LIN {X -0.084,Y -142.879,Z 263.170,A 0.000,B 0.000,C 90.000,E1 210.669} C_DIS
LIN {X -0.027,Y -141.496,Z 263.150,A 0.000,B 0.000,C 90.000,E1 206.950} C_DIS
LIN {X 0.023,Y -139.387,Z 263.114,A 0.000,B 0.000,C 90.000,E1 200.429} C_DIS
LIN {X 0.010,Y -138.843,Z 263.098,A 0.000,B 0.000,C 90.000,E1 197.638} C_DIS
LIN {X -0.066,Y -138.354,Z 263.056,A 0.000,B 0.000,C 90.000,E1 190.197} C_DIS
LIN {X 0.067,Y -139.519,Z 263.005,A 0.000,B 0.000,C 90.000,E1 180.802} C_DIS
LIN {X 0.007,Y -141.176,Z 262.974,A 0.000,B 0.000,C 90.000,E1 175.241} C_DIS
LIN {X -0.021,Y -142.555,Z 262.958,A 0.000,B 0.000,C 90.000,E1 172.470} C_DIS
LIN {X 0.046,Y -144.834,Z 262.932,A 0.000,B 0.000,C 90.000,E1 167.825} C_DIS
LIN {X 0.031,Y -147.457,Z 262.912,A 0.000,B 0.000,C 90.000,E1 164.157} C_DIS
LIN {X -0.082,Y -150.039,Z 262.892,A 0.000,B 0.000,C 90.000,E1 160.550} C_DIS
LIN {X -0.076,Y -153.380,Z 262.872,A 0.000,B 0.000,C 90.000,E1 156.922} C_DIS
LIN {X -0.029,Y -155.912,Z 262.857,A 0.000,B 0.000,C 90.000,E1 154.204} C_DIS
LIN {X 0.087,Y -159.775,Z 262.837,A 0.000,B 0.000,C 90.000,E1 150.589} C_DIS
LIN {X -0.066,Y -162.015,Z 262.827,A 0.000,B 0.000,C 90.000,E1 148.869} C_DIS
LIN {X 0.048,Y -166.209,Z 262.807,A 0.000,B 0.000,C 90.000,E1 145.308} C_DIS
LIN {X 0.049,Y -171.225,Z 262.788,A 0.000,B 0.000,C 90.000,E1 141.823} C_DIS
LIN {X -0.026,Y -176.111,Z 262.769,A 0.000,B 0.000,C 90.000,E1 138.405} C_DIS
LIN {X 0.090,Y -180.375,Z 262.755,A 0.000,B 0.000,C 90.000,E1 135.810} C_DIS
LIN {X 0.067,Y -185.783,Z 262.736,A 0.000,B 0.000,C 90.000,E1 132.447} C_DIS
LIN {X 0.000,Y -190.399,Z 262.722,A 0.000,B 0.000,C 90.000,E1 129.967} C_DIS
LIN {X 0.016,Y -197.723,Z 262.699,A 0.000,B 0.000,C 90.000,E1 125.851} C_DIS
LIN {X -0.060,Y -200.971,Z 262.690,A 0.000,B 0.000,C 90.000,E1 124.246} C_DIS
LIN {X 0.078,Y -203.895,Z 262.681,A 0.000,B 0.000,C 90.000,E1 122.546} C_DIS
LIN {X 0.064,Y -306.288,Z 262.681,A 0.000,B 0.000,C 90.000,E1 122.546} C_DIS
LIN {X 0.009,Y -307.336,Z 262.681,A 0.000,B 0.000,C 90.000,E1 122.546} C_DIS
LIN {X 0.131,Y -312.237,Z 262.680,A 0.000,B 0.000,C 90.000,E1 122.339} C_DIS
LIN {X -0.178,Y -314.694,Z 262.679,A 0.000,B 0.000,C 90.000,E1 122.212} C_DIS
LIN {X 0.068,Y -318.006,Z 262.677,A 0.000,B 0.000,C 90.000,E1 121.799} C_DIS
LIN {X -0.031,Y -319.961,Z 262.675,A 0.000,B 0.000,C 90.000,E1 121.514} C_DIS
LIN {X -0.026,Y -321.496,Z 262.673,A 0.000,B 0.000,C 90.000,E1 121.209} C_DIS
LIN {X 0.054,Y -335.561,Z 262.654,A 0.000,B 0.000,C 90.000,E1 117.719} C_DIS
LIN {X -0.033,Y -348.593,Z 262.639,A 0.000,B 0.000,C 90.000,E1 114.951} C_DIS
LIN {X 0.068,Y -361.495,Z 262.625,A 0.000,B 0.000,C 90.000,E1 112.514} C_DIS
LIN {X -0.119,Y -375.736,Z 262.612,A 0.000,B 0.000,C 90.000,E1 110.174} C_DIS
LIN {X 0.152,Y -391.421,Z 262.599,A 0.000,B 0.000,C 90.000,E1 107.819} C_DIS
LIN {X -0.164,Y -408.665,Z 262.587,A 0.000,B 0.000,C 90.000,E1 105.607} C_DIS
LIN {X -0.185,Y -427.600,Z 262.574,A 0.000,B 0.000,C 90.000,E1 103.411} C_DIS
LIN {X 0.123,Y -447.711,Z 262.563,A 0.000,B 0.000,C 90.000,E1 101.299} C_DIS
LIN {X -0.145,Y -468.376,Z 262.552,A 0.000,B 0.000,C 90.000,E1 99.434} C_DIS
LIN {X 0.024,Y -492.186,Z 262.542,A 0.000,B 0.000,C 90.000,E1 97.466} C_DIS
LIN {X -0.023,Y -502.840,Z 262.537,A 0.000,B 0.000,C 90.000,E1 96.663} C_DIS
LIN {X -0.205,Y -504.840,Z 262.536,A 0.000,B 0.000,C 90.000,E1 96.486} C_DIS
LIN {X 0.199,Y -506.671,Z 262.535,A 0.000,B 0.000,C 90.000,E1 96.201} C_DIS
LIN {X 0.157,Y -508.048,Z 262.533,A 0.000,B 0.000,C 90.000,E1 95.967} C_DIS
LIN {X -0.073,Y -509.799,Z 262.531,A 0.000,B 0.000,C 90.000,E1 95.511} C_DIS
LIN {X -0.244,Y -510.440,Z 262.528,A 0.000,B 0.000,C 90.000,E1 95.049} C_DIS
LIN {X 0.101,Y -510.071,Z 262.525,A 0.000,B 0.000,C 90.000,E1 94.531} C_DIS
LIN {X -0.099,Y -508.627,Z 262.523,A 0.000,B 0.000,C 90.000,E1 94.073} C_DIS
LIN {X -0.163,Y -507.423,Z 262.521,A 0.000,B 0.000,C 90.000,E1 93.841} C_DIS
LIN {X 0.138,Y -503.972,Z 262.519,A 0.000,B 0.000,C 90.000,E1 93.326} C_DIS
LIN {X -0.166,Y -498.128,Z 262.515,A 0.000,B 0.000,C 90.000,E1 92.636} C_DIS
LIN {X 0.187,Y -487.577,Z 262.508,A 0.000,B 0.000,C 90.000,E1 91.375} C_DIS
LIN {X -0.069,Y -466.396,Z 262.494,A 0.000,B 0.000,C 90.000,E1 88.912} C_DIS
LIN {X 0.086,Y -451.279,Z 262.483,A 0.000,B 0.000,C 90.000,E1 86.846} C_DIS
LIN {X 0.022,Y -432.472,Z 262.467,A 0.000,B 0.000,C 90.000,E1 83.970} C_DIS
LIN {X 0.219,Y -416.903,Z 262.452,A 0.000,B 0.000,C 90.000,E1 81.254} C_DIS
LIN {X -0.015,Y -404.099,Z 262.438,A 0.000,B 0.000,C 90.000,E1 78.814} C_DIS
LIN {X -0.040,Y -391.301,Z 262.424,A 0.000,B 0.000,C 90.000,E1 76.297} C_DIS
LIN {X -0.128,Y -378.784,Z 262.410,A 0.000,B 0.000,C 90.000,E1 73.740} C_DIS
LIN {X -0.060,Y -367.611,Z 262.397,A 0.000,B 0.000,C 90.000,E1 71.402} C_DIS
LIN {X -0.032,Y -356.629,Z 262.383,A 0.000,B 0.000,C 90.000,E1 69.028} C_DIS
LIN {X 0.187,Y -342.383,Z 262.365,A 0.000,B 0.000,C 90.000,E1 65.665} C_DIS
LIN {X -0.064,Y -330.397,Z 262.348,A 0.000,B 0.000,C 90.000,E1 62.615} C_DIS
LIN {X -0.055,Y -319.220,Z 262.330,A 0.000,B 0.000,C 90.000,E1 59.459} C_DIS
LIN {X -0.178,Y -310.444,Z 262.316,A 0.000,B 0.000,C 90.000,E1 56.914} C_DIS
LIN {X -0.009,Y -299.955,Z 262.298,A 0.000,B 0.000,C 90.000,E1 53.623} C_DIS
LIN {X 0.093,Y -293.735,Z 262.287,A 0.000,B 0.000,C 90.000,E1 51.618} C_DIS
LIN {X 0.103,Y -285.428,Z 262.272,A 0.000,B 0.000,C 90.000,E1 48.933} C_DIS
LIN {X -0.121,Y -275.297,Z 262.253,A 0.000,B 0.000,C 90.000,E1 45.567} C_DIS
LIN {X -0.020,Y -267.641,Z 262.238,A 0.000,B 0.000,C 90.000,E1 42.771} C_DIS
LIN {X 0.090,Y -260.135,Z 262.222,A 0.000,B 0.000,C 90.000,E1 39.930} C_DIS
LIN {X 0.007,Y -254.382,Z 262.210,A 0.000,B 0.000,C 90.000,E1 37.810} C_DIS
LIN {X 0.016,Y -248.606,Z 262.198,A 0.000,B 0.000,C 90.000,E1 35.644} C_DIS
LIN {X -0.117,Y -240.937,Z 262.182,A 0.000,B 0.000,C 90.000,E1 32.752} C_DIS
LIN {X 0.033,Y -231.734,Z 262.161,A 0.000,B 0.000,C 90.000,E1 28.999} C_DIS
LIN {X 0.028,Y -225.126,Z 262.144,A 0.000,B 0.000,C 90.000,E1 25.976} C_DIS
LIN {X 0.076,Y -219.297,Z 262.127,A 0.000,B 0.000,C 90.000,E1 22.898} C_DIS
LIN {X 0.002,Y -212.842,Z 262.106,A 0.000,B 0.000,C 90.000,E1 19.033} C_DIS
LIN {X 0.068,Y -207.446,Z 262.084,A 0.000,B 0.000,C 90.000,E1 15.079} C_DIS
LIN {X -0.045,Y -202.998,Z 262.062,A 0.000,B 0.000,C 90.000,E1 11.130} C_DIS
LIN {X -0.087,Y -199.578,Z 262.039,A 0.000,B 0.000,C 90.000,E1 7.125} C_DIS
LIN {X -0.009,Y -196.386,Z 262.008,A 0.000,B 0.000,C 90.000,E1 1.432} C_DIS
LIN {X 0.078,Y -197.440,Z 261.920,A 0.000,B 0.000,C 90.000,E1 345.644} C_DIS
LIN {X 0.059,Y -200.766,Z 261.893,A 0.000,B 0.000,C 90.000,E1 340.786} C_DIS
LIN {X -0.056,Y -204.789,Z 261.871,A 0.000,B 0.000,C 90.000,E1 336.794} C_DIS
LIN {X -0.009,Y -209.928,Z 261.849,A 0.000,B 0.000,C 90.000,E1 332.794} C_DIS
LIN {X -0.070,Y -216.233,Z 261.827,A 0.000,B 0.000,C 90.000,E1 328.869} C_DIS
LIN {X 0.059,Y -222.165,Z 261.810,A 0.000,B 0.000,C 90.000,E1 325.722} C_DIS
LIN {X 0.102,Y -228.969,Z 261.793,A 0.000,B 0.000,C 90.000,E1 322.637} C_DIS
LIN {X 0.006,Y -237.487,Z 261.774,A 0.000,B 0.000,C 90.000,E1 319.256} C_DIS
LIN {X 0.112,Y -246.994,Z 261.755,A 0.000,B 0.000,C 90.000,E1 315.891} C_DIS
LIN {X 0.155,Y -257.496,Z 261.737,A 0.000,B 0.000,C 90.000,E1 312.609} C_DIS
LIN {X -0.005,Y -269.138,Z 261.719,A 0.000,B 0.000,C 90.000,E1 309.439} C_DIS
LIN {X 0.042,Y -282.107,Z 261.702,A 0.000,B 0.000,C 90.000,E1 306.297} C_DIS
LIN {X 0.039,Y -295.069,Z 261.687,A 0.000,B 0.000,C 90.000,E1 303.579} C_DIS
LIN {X -0.016,Y -305.748,Z 261.676,A 0.000,B 0.000,C 90.000,E1 301.592} C_DIS
LIN {X -0.065,Y -321.117,Z 261.661,A 0.000,B 0.000,C 90.000,E1 298.999} C_DIS
LIN {X -0.072,Y -339.487,Z 261.645,A 0.000,B 0.000,C 90.000,E1 296.155} C_DIS
LIN {X 0.084,Y -351.911,Z 261.635,A 0.000,B 0.000,C 90.000,E1 294.283} C_DIS
LIN {X 0.167,Y -364.417,Z 261.625,A 0.000,B 0.000,C 90.000,E1 292.461} C_DIS
LIN {X 0.079,Y -381.335,Z 261.612,A 0.000,B 0.000,C 90.000,E1 290.120} C_DIS
LIN {X -0.025,Y -396.501,Z 261.601,A 0.000,B 0.000,C 90.000,E1 288.127} C_DIS
LIN {X -0.114,Y -407.339,Z 261.593,A 0.000,B 0.000,C 90.000,E1 286.732} C_DIS
LIN {X 0.095,Y -422.232,Z 261.582,A 0.000,B 0.000,C 90.000,E1 284.773} C_DIS
LIN {X -0.012,Y -430.385,Z 261.576,A 0.000,B 0.000,C 90.000,E1 283.703} C_DIS
LIN {X -0.129,Y -437.902,Z 261.570,A 0.000,B 0.000,C 90.000,E1 282.647} C_DIS
LIN {X -0.159,Y -444.744,Z 261.564,A 0.000,B 0.000,C 90.000,E1 281.591} C_DIS
LIN {X -0.144,Y -454.217,Z 261.556,A 0.000,B 0.000,C 90.000,E1 280.018} C_DIS
LIN {X 0.138,Y -461.619,Z 261.548,A 0.000,B 0.000,C 90.000,E1 278.690} C_DIS
LIN {X 0.150,Y -468.491,Z 261.541,A 0.000,B 0.000,C 90.000,E1 277.409} C_DIS
LIN {X -0.133,Y -473.614,Z 261.536,A 0.000,B 0.000,C 90.000,E1 276.429} C_DIS
LIN {X -0.217,Y -477.139,Z 261.531,A 0.000,B 0.000,C 90.000,E1 275.682} C_DIS
LIN {X -0.079,Y -479.157,Z 261.529,A 0.000,B 0.000,C 90.000,E1 275.163} C_DIS
LIN {X 0.065,Y -480.938,Z 261.526,A 0.000,B 0.000,C 90.000,E1 274.645} C_DIS
LIN {X 0.185,Y -482.344,Z 261.523,A 0.000,B 0.000,C 90.000,E1 274.131} C_DIS
LIN {X -0.132,Y -483.499,Z 261.520,A 0.000,B 0.000,C 90.000,E1 273.669} C_DIS
LIN {X 0.012,Y -484.296,Z 261.518,A 0.000,B 0.000,C 90.000,E1 273.154} C_DIS
LIN {X 0.188,Y -484.741,Z 261.515,A 0.000,B 0.000,C 90.000,E1 272.636} C_DIS
LIN {X 0.041,Y -485.008,Z 261.509,A 0.000,B 0.000,C 90.000,E1 271.661} C_DIS
LIN {X 0.203,Y -484.935,Z 261.507,A 0.000,B 0.000,C 90.000,E1 271.146} C_DIS
LIN {X -0.117,Y -484.681,Z 261.504,A 0.000,B 0.000,C 90.000,E1 270.688} C_DIS
LIN {X 0.049,Y -484.046,Z 261.501,A 0.000,B 0.000,C 90.000,E1 270.172} C_DIS
LIN {X 0.212,Y -483.060,Z 261.498,A 0.000,B 0.000,C 90.000,E1 269.656} C_DIS
LIN {X -0.112,Y -481.501,Z 261.495,A 0.000,B 0.000,C 90.000,E1 269.198} C_DIS
LIN {X 0.040,Y -479.301,Z 261.493,A 0.000,B 0.000,C 90.000,E1 268.682} C_DIS
LIN {X 0.175,Y -476.392,Z 261.490,A 0.000,B 0.000,C 90.000,E1 268.167} C_DIS
LIN {X -0.164,Y -472.714,Z 261.487,A 0.000,B 0.000,C 90.000,E1 267.707} C_DIS
LIN {X -0.063,Y -468.210,Z 261.484,A 0.000,B 0.000,C 90.000,E1 267.192} C_DIS
LIN {X 0.205,Y -465.592,Z 261.483,A 0.000,B 0.000,C 90.000,E1 266.906} C_DIS
LIN {X 0.034,Y -462.649,Z 261.482,A 0.000,B 0.000,C 90.000,E1 266.674} C_DIS
LIN {X 0.083,Y -456.463,Z 261.479,A 0.000,B 0.000,C 90.000,E1 266.216} C_DIS
LIN {X -0.104,Y -453.228,Z 261.478,A 0.000,B 0.000,C 90.000,E1 266.045} C_DIS
LIN {X 0.193,Y -449.532,Z 261.477,A 0.000,B 0.000,C 90.000,E1 265.812} C_DIS
LIN {X -0.132,Y -445.984,Z 261.476,A 0.000,B 0.000,C 90.000,E1 265.698} C_DIS
LIN {X -0.011,Y -441.741,Z 261.475,A 0.000,B 0.000,C 90.000,E1 265.527} C_DIS
LIN {X -0.002,Y -437.789,Z 261.475,A 0.000,B 0.000,C 90.000,E1 265.412} C_DIS
LIN {X 0.008,Y -432.446,Z 261.474,A 0.000,B 0.000,C 90.000,E1 265.298} C_DIS
LIN {X 0.144,Y -425.453,Z 261.473,A 0.000,B 0.000,C 90.000,E1 265.179} C_DIS
LIN {X -0.163,Y -418.203,Z 261.473,A 0.000,B 0.000,C 90.000,E1 265.179} C_DIS
LIN {X 0.084,Y -180.889,Z 261.473,A 0.000,B 0.000,C 90.000,E1 265.122} C_DIS
LIN {X -0.014,Y -179.001,Z 261.445,A 0.000,B 0.000,C 90.000,E1 260.038} C_DIS
LIN {X 0.079,Y -178.598,Z 261.440,A 0.000,B 0.000,C 90.000,E1 259.162} C_DIS
LIN {X -0.027,Y -175.650,Z 261.412,A 0.000,B 0.000,C 90.000,E1 254.102} C_DIS
LIN {X -0.021,Y -172.368,Z 261.388,A 0.000,B 0.000,C 90.000,E1 249.826} C_DIS
LIN {X -0.007,Y -171.160,Z 261.378,A 0.000,B 0.000,C 90.000,E1 248.103} C_DIS
LIN {X 0.037,Y -167.459,Z 261.354,A 0.000,B 0.000,C 90.000,E1 243.768} C_DIS
LIN {X -0.030,Y -166.856,Z 261.350,A 0.000,B 0.000,C 90.000,E1 242.922} C_DIS
LIN {X 0.035,Y -162.841,Z 261.325,A 0.000,B 0.000,C 90.000,E1 238.535} C_DIS
LIN {X 0.010,Y -161.524,Z 261.315,A 0.000,B 0.000,C 90.000,E1 236.786} C_DIS
LIN {X 0.050,Y -157.524,Z 261.291,A 0.000,B 0.000,C 90.000,E1 232.351} C_DIS
LIN {X -0.017,Y -155.548,Z 261.276,A 0.000,B 0.000,C 90.000,E1 229.703} C_DIS
LIN {X -0.082,Y -151.840,Z 261.251,A 0.000,B 0.000,C 90.000,E1 225.243} C_DIS
LIN {X -0.068,Y -150.058,Z 261.236,A 0.000,B 0.000,C 90.000,E1 222.528} C_DIS
LIN {X -0.033,Y -146.870,Z 261.211,A 0.000,B 0.000,C 90.000,E1 217.971} C_DIS
LIN {X -0.044,Y -145.455,Z 261.196,A 0.000,B 0.000,C 90.000,E1 215.231} C_DIS
LIN {X 0.070,Y -142.871,Z 261.170,A 0.000,B 0.000,C 90.000,E1 210.590} C_DIS
LIN {X -0.005,Y -141.489,Z 261.150,A 0.000,B 0.000,C 90.000,E1 206.924} C_DIS
LIN {X -0.020,Y -139.384,Z 261.113,A 0.000,B 0.000,C 90.000,E1 200.429} C_DIS
LIN {X -0.031,Y -138.839,Z 261.098,A 0.000,B 0.000,C 90.000,E1 197.638} C_DIS
LIN {X 0.029,Y -138.353,Z 261.056,A 0.000,B 0.000,C 90.000,E1 190.141} C_DIS
LIN {X 0.025,Y -139.521,Z 261.005,A 0.000,B 0.000,C 90.000,E1 180.802} C_DIS
LIN {X -0.035,Y -141.184,Z 260.973,A 0.000,B 0.000,C 90.000,E1 175.241} C_DIS
LIN {X -0.064,Y -142.562,Z 260.958,A 0.000,B 0.000,C 90.000,E1 172.470} C_DIS
LIN {X 0.002,Y -144.844,Z 260.932,A 0.000,B 0.000,C 90.000,E1 167.825} C_DIS
LIN {X -0.012,Y -147.469,Z 260.912,A 0.000,B 0.000,C 90.000,E1 164.157} C_DIS
LIN {X 0.016,Y -150.054,Z 260.892,A 0.000,B 0.000,C 90.000,E1 160.496} C_DIS
LIN {X 0.020,Y -153.397,Z 260.872,A 0.000,B 0.000,C 90.000,E1 156.869} C_DIS
LIN {X 0.067,Y -155.927,Z 260.857,A 0.000,B 0.000,C 90.000,E1 154.152} C_DIS
LIN {X 0.041,Y -159.795,Z 260.837,A 0.000,B 0.000,C 90.000,E1 150.589} C_DIS
LIN {X 0.026,Y -162.035,Z 260.827,A 0.000,B 0.000,C 90.000,E1 148.820} C_DIS
LIN {X 0.001,Y -166.231,Z 260.807,A 0.000,B 0.000,C 90.000,E1 145.308} C_DIS
LIN {X 0.002,Y -171.247,Z 260.788,A 0.000,B 0.000,C 90.000,E1 141.823} C_DIS
LIN {X -0.075,Y -176.136,Z 260.769,A 0.000,B 0.000,C 90.000,E1 138.405} C_DIS
LIN {X 0.041,Y -180.403,Z 260.755,A 0.000,B 0.000,C 90.000,E1 135.810} C_DIS
LIN {X 0.017,Y -185.810,Z 260.736,A 0.000,B 0.000,C 90.000,E1 132.447} C_DIS
LIN {X 0.071,Y -190.429,Z 260.722,A 0.000,B 0.000,C 90.000,E1 129.930} C_DIS
LIN {X -0.037,Y -197.753,Z 260.699,A 0.000,B 0.000,C 90.000,E1 125.851} C_DIS
LIN {X 0.054,Y -200.996,Z 260.690,A 0.000,B 0.000,C 90.000,E1 124.199} C_DIS
LIN {X 0.031,Y -204.009,Z 260.681,A 0.000,B 0.000,C 90.000,E1 122.498} C_DIS
LIN {X -0.005,Y -307.390,Z 260.681,A 0.000,B 0.000,C 90.000,E1 122.498} C_DIS
LIN {X 0.002,Y -308.854,Z 260.680,A 0.000,B 0.000,C 90.000,E1 122.467} C_DIS
LIN {X 0.047,Y -312.597,Z 260.679,A 0.000,B 0.000,C 90.000,E1 122.291} C_DIS
LIN {X -0.007,Y -314.817,Z 260.678,A 0.000,B 0.000,C 90.000,E1 122.133} C_DIS
LIN {X -0.014,Y -317.903,Z 260.677,A 0.000,B 0.000,C 90.000,E1 121.799} C_DIS
LIN {X 0.186,Y -319.892,Z 260.675,A 0.000,B 0.000,C 90.000,E1 121.465} C_DIS
LIN {X -0.052,Y -321.453,Z 260.673,A 0.000,B 0.000,C 90.000,E1 121.209} C_DIS
LIN {X -0.175,Y -331.546,Z 260.659,A 0.000,B 0.000,C 90.000,E1 118.693} C_DIS
LIN {X 0.085,Y -344.080,Z 260.644,A 0.000,B 0.000,C 90.000,E1 115.848} C_DIS
LIN {X -0.106,Y -356.507,Z 260.630,A 0.000,B 0.000,C 90.000,E1 113.439} C_DIS
LIN {X -0.080,Y -370.235,Z 260.617,A 0.000,B 0.000,C 90.000,E1 111.046} C_DIS
LIN {X -0.180,Y -385.367,Z 260.604,A 0.000,B 0.000,C 90.000,E1 108.725} C_DIS
LIN {X -0.156,Y -402.016,Z 260.591,A 0.000,B 0.000,C 90.000,E1 106.441} C_DIS
LIN {X 0.071,Y -420.304,Z 260.579,A 0.000,B 0.000,C 90.000,E1 104.189} C_DIS
LIN {X 0.030,Y -440.104,Z 260.567,A 0.000,B 0.000,C 90.000,E1 102.063} C_DIS
LIN {X 0.173,Y -460.571,Z 260.556,A 0.000,B 0.000,C 90.000,E1 100.084} C_DIS
LIN {X -0.112,Y -484.215,Z 260.545,A 0.000,B 0.000,C 90.000,E1 98.106} C_DIS
LIN {X -0.058,Y -502.890,Z 260.537,A 0.000,B 0.000,C 90.000,E1 96.663} C_DIS
LIN {X 0.262,Y -504.933,Z 260.536,A 0.000,B 0.000,C 90.000,E1 96.429} C_DIS
LIN {X 0.192,Y -506.782,Z 260.535,A 0.000,B 0.000,C 90.000,E1 96.201} C_DIS
LIN {X 0.176,Y -508.177,Z 260.533,A 0.000,B 0.000,C 90.000,E1 95.967} C_DIS
LIN {X -0.053,Y -509.984,Z 260.531,A 0.000,B 0.000,C 90.000,E1 95.511} C_DIS
LIN {X -0.224,Y -510.666,Z 260.528,A 0.000,B 0.000,C 90.000,E1 95.049} C_DIS
LIN {X 0.122,Y -510.338,Z 260.525,A 0.000,B 0.000,C 90.000,E1 94.531} C_DIS
LIN {X -0.077,Y -508.947,Z 260.523,A 0.000,B 0.000,C 90.000,E1 94.073} C_DIS
LIN {X -0.140,Y -507.775,Z 260.521,A 0.000,B 0.000,C 90.000,E1 93.841} C_DIS
LIN {X 0.163,Y -504.368,Z 260.519,A 0.000,B 0.000,C 90.000,E1 93.326} C_DIS
LIN {X -0.138,Y -498.540,Z 260.515,A 0.000,B 0.000,C 90.000,E1 92.636} C_DIS
LIN {X -0.127,Y -490.145,Z 260.509,A 0.000,B 0.000,C 90.000,E1 91.661} C_DIS
LIN {X -0.026,Y -466.770,Z 260.494,A 0.000,B 0.000,C 90.000,E1 88.912} C_DIS
LIN {X -0.107,Y -453.453,Z 260.484,A 0.000,B 0.000,C 90.000,E1 87.135} C_DIS
LIN {X 0.164,Y -436.097,Z 260.470,A 0.000,B 0.000,C 90.000,E1 84.489} C_DIS
LIN {X 0.134,Y -418.677,Z 260.453,A 0.000,B 0.000,C 90.000,E1 81.546} C_DIS
LIN {X 0.055,Y -404.388,Z 260.438,A 0.000,B 0.000,C 90.000,E1 78.814} C_DIS
LIN {X 0.036,Y -391.568,Z 260.424,A 0.000,B 0.000,C 90.000,E1 76.297} C_DIS
LIN {X -0.047,Y -379.079,Z 260.410,A 0.000,B 0.000,C 90.000,E1 73.740} C_DIS
LIN {X 0.026,Y -367.931,Z 260.397,A 0.000,B 0.000,C 90.000,E1 71.402} C_DIS
LIN {X 0.059,Y -356.974,Z 260.384,A 0.000,B 0.000,C 90.000,E1 69.028} C_DIS
LIN {X -0.026,Y -342.765,Z 260.365,A 0.000,B 0.000,C 90.000,E1 65.717} C_DIS
LIN {X 0.043,Y -330.801,Z 260.348,A 0.000,B 0.000,C 90.000,E1 62.615} C_DIS
LIN {X 0.067,Y -319.624,Z 260.330,A 0.000,B 0.000,C 90.000,E1 59.459} C_DIS
LIN {X -0.022,Y -310.881,Z 260.316,A 0.000,B 0.000,C 90.000,E1 56.914} C_DIS
LIN {X 0.154,Y -300.371,Z 260.298,A 0.000,B 0.000,C 90.000,E1 53.623} C_DIS
LIN {X 0.030,Y -294.159,Z 260.287,A 0.000,B 0.000,C 90.000,E1 51.662} C_DIS
LIN {X -0.127,Y -285.836,Z 260.272,A 0.000,B 0.000,C 90.000,E1 49.013} C_DIS
LIN {X 0.059,Y -275.703,Z 260.253,A 0.000,B 0.000,C 90.000,E1 45.567} C_DIS
LIN {X -0.033,Y -268.039,Z 260.238,A 0.000,B 0.000,C 90.000,E1 42.813} C_DIS
LIN {X -0.087,Y -260.528,Z 260.222,A 0.000,B 0.000,C 90.000,E1 40.011} C_DIS
LIN {X -0.002,Y -254.769,Z 260.210,A 0.000,B 0.000,C 90.000,E1 37.855} C_DIS
LIN {X -0.049,Y -247.083,Z 260.194,A 0.000,B 0.000,C 90.000,E1 34.978} C_DIS
LIN {X 0.121,Y -239.463,Z 260.178,A 0.000,B 0.000,C 90.000,E1 32.005} C_DIS
LIN {X -0.080,Y -232.152,Z 260.161,A 0.000,B 0.000,C 90.000,E1 29.077} C_DIS
LIN {X 0.033,Y -225.527,Z 260.145,A 0.000,B 0.000,C 90.000,E1 26.027} C_DIS
LIN {X 0.085,Y -219.685,Z 260.128,A 0.000,B 0.000,C 90.000,E1 22.950} C_DIS
LIN {X 0.018,Y -213.215,Z 260.106,A 0.000,B 0.000,C 90.000,E1 19.087} C_DIS
LIN {X -0.110,Y -207.817,Z 260.084,A 0.000,B 0.000,C 90.000,E1 15.190} C_DIS
LIN {X -0.015,Y -203.339,Z 260.062,A 0.000,B 0.000,C 90.000,E1 11.186} C_DIS
LIN {X -0.050,Y -199.886,Z 260.040,A 0.000,B 0.000,C 90.000,E1 7.182} C_DIS
LIN {X 0.003,Y -196.350,Z 260.004,A 0.000,B 0.000,C 90.000,E1 0.688} C_DIS
LIN {X 0.080,Y -197.248,Z 259.925,A 0.000,B 0.000,C 90.000,E1 346.464} C_DIS
LIN {X -0.061,Y -200.306,Z 259.898,A 0.000,B 0.000,C 90.000,E1 341.638} C_DIS
LIN {X -0.001,Y -204.069,Z 259.876,A 0.000,B 0.000,C 90.000,E1 337.592} C_DIS
LIN {X 0.035,Y -208.988,Z 259.853,A 0.000,B 0.000,C 90.000,E1 333.589} C_DIS
LIN {X -0.061,Y -215.090,Z 259.831,A 0.000,B 0.000,C 90.000,E1 329.665} C_DIS
LIN {X 0.104,Y -220.800,Z 259.814,A 0.000,B 0.000,C 90.000,E1 326.501} C_DIS
LIN {X 0.111,Y -227.432,Z 259.797,A 0.000,B 0.000,C 90.000,E1 323.417} C_DIS
LIN {X -0.133,Y -234.790,Z 259.780,A 0.000,B 0.000,C 90.000,E1 320.436} C_DIS
LIN {X -0.107,Y -243.924,Z 259.761,A 0.000,B 0.000,C 90.000,E1 317.067} C_DIS
LIN {X 0.015,Y -254.095,Z 259.743,A 0.000,B 0.000,C 90.000,E1 313.743} C_DIS
LIN {X -0.092,Y -265.335,Z 259.725,A 0.000,B 0.000,C 90.000,E1 310.539} C_DIS
LIN {X 0.001,Y -277.812,Z 259.708,A 0.000,B 0.000,C 90.000,E1 307.363} C_DIS
LIN {X 0.078,Y -288.604,Z 259.694,A 0.000,B 0.000,C 90.000,E1 304.945} C_DIS
LIN {X -0.086,Y -302.262,Z 259.679,A 0.000,B 0.000,C 90.000,E1 302.291} C_DIS
LIN {X 0.000,Y -319.334,Z 259.663,A 0.000,B 0.000,C 90.000,E1 299.333} C_DIS
LIN {X 0.079,Y -339.615,Z 259.645,A 0.000,B 0.000,C 90.000,E1 296.155} C_DIS
LIN {X -0.078,Y -352.006,Z 259.635,A 0.000,B 0.000,C 90.000,E1 294.335} C_DIS
LIN {X -0.004,Y -364.464,Z 259.625,A 0.000,B 0.000,C 90.000,E1 292.514} C_DIS
LIN {X -0.104,Y -381.346,Z 259.612,A 0.000,B 0.000,C 90.000,E1 290.174} C_DIS
LIN {X -0.054,Y -398.637,Z 259.599,A 0.000,B 0.000,C 90.000,E1 287.873} C_DIS
LIN {X 0.163,Y -409.395,Z 259.591,A 0.000,B 0.000,C 90.000,E1 286.441} C_DIS
LIN {X -0.122,Y -422.118,Z 259.582,A 0.000,B 0.000,C 90.000,E1 284.828} C_DIS
LIN {X 0.080,Y -430.248,Z 259.576,A 0.000,B 0.000,C 90.000,E1 283.716} C_DIS
LIN {X 0.066,Y -437.738,Z 259.570,A 0.000,B 0.000,C 90.000,E1 282.647} C_DIS
LIN {X 0.037,Y -444.571,Z 259.564,A 0.000,B 0.000,C 90.000,E1 281.591} C_DIS
LIN {X 0.053,Y -454.038,Z 259.556,A 0.000,B 0.000,C 90.000,E1 280.018} C_DIS
LIN {X -0.120,Y -461.433,Z 259.548,A 0.000,B 0.000,C 90.000,E1 278.746} C_DIS
LIN {X -0.117,Y -468.316,Z 259.541,A 0.000,B 0.000,C 90.000,E1 277.466} C_DIS
LIN {X -0.142,Y -474.637,Z 259.534,A 0.000,B 0.000,C 90.000,E1 276.201} C_DIS
LIN {X -0.165,Y -478.001,Z 259.530,A 0.000,B 0.000,C 90.000,E1 275.448} C_DIS
LIN {X -0.210,Y -480.795,Z 259.526,A 0.000,B 0.000,C 90.000,E1 274.702} C_DIS
LIN {X -0.094,Y -482.249,Z 259.523,A 0.000,B 0.000,C 90.000,E1 274.188} C_DIS
LIN {X 0.071,Y -483.416,Z 259.520,A 0.000,B 0.000,C 90.000,E1 273.669} C_DIS
LIN {X 0.214,Y -484.213,Z 259.518,A 0.000,B 0.000,C 90.000,E1 273.154} C_DIS
LIN {X -0.093,Y -484.705,Z 259.515,A 0.000,B 0.000,C 90.000,E1 272.694} C_DIS
LIN {X 0.242,Y -485.059,Z 259.509,A 0.000,B 0.000,C 90.000,E1 271.661} C_DIS
LIN {X -0.079,Y -485.030,Z 259.507,A 0.000,B 0.000,C 90.000,E1 271.203} C_DIS
LIN {X 0.085,Y -484.782,Z 259.504,A 0.000,B 0.000,C 90.000,E1 270.688} C_DIS
LIN {X -0.234,Y -484.227,Z 259.501,A 0.000,B 0.000,C 90.000,E1 270.229} C_DIS
LIN {X -0.069,Y -483.221,Z 259.498,A 0.000,B 0.000,C 90.000,E1 269.714} C_DIS
LIN {X 0.091,Y -481.668,Z 259.496,A 0.000,B 0.000,C 90.000,E1 269.198} C_DIS
LIN {X -0.236,Y -479.526,Z 259.493,A 0.000,B 0.000,C 90.000,E1 268.740} C_DIS
LIN {X -0.093,Y -476.672,Z 259.490,A 0.000,B 0.000,C 90.000,E1 268.224} C_DIS
LIN {X 0.044,Y -473.033,Z 259.487,A 0.000,B 0.000,C 90.000,E1 267.707} C_DIS
LIN {X -0.140,Y -470.944,Z 259.486,A 0.000,B 0.000,C 90.000,E1 267.478} C_DIS
LIN {X -0.052,Y -465.992,Z 259.483,A 0.000,B 0.000,C 90.000,E1 266.963} C_DIS
LIN {X -0.217,Y -460.211,Z 259.480,A 0.000,B 0.000,C 90.000,E1 266.502} C_DIS
LIN {X 0.039,Y -453.842,Z 259.478,A 0.000,B 0.000,C 90.000,E1 266.045} C_DIS
LIN {X -0.130,Y -450.177,Z 259.477,A 0.000,B 0.000,C 90.000,E1 265.869} C_DIS
LIN {X -0.025,Y -446.756,Z 259.476,A 0.000,B 0.000,C 90.000,E1 265.698} C_DIS
LIN {X 0.077,Y -442.552,Z 259.475,A 0.000,B 0.000,C 90.000,E1 265.527} C_DIS
LIN {X 0.065,Y -438.690,Z 259.475,A 0.000,B 0.000,C 90.000,E1 265.412} C_DIS
LIN {X -0.054,Y -429.430,Z 259.474,A 0.000,B 0.000,C 90.000,E1 265.241} C_DIS
LIN {X 0.141,Y -419.581,Z 259.473,A 0.000,B 0.000,C 90.000,E1 265.122} C_DIS
LIN {X 0.028,Y -180.887,Z 259.473,A 0.000,B 0.000,C 90.000,E1 265.122} C_DIS
LIN {X -0.075,Y -178.997,Z 259.445,A 0.000,B 0.000,C 90.000,E1 260.038} C_DIS
LIN {X 0.019,Y -178.584,Z 259.440,A 0.000,B 0.000,C 90.000,E1 259.162} C_DIS
LIN {X -0.088,Y -175.636,Z 259.412,A 0.000,B 0.000,C 90.000,E1 254.102} C_DIS
LIN {X -0.021,Y -172.356,Z 259.388,A 0.000,B 0.000,C 90.000,E1 249.806} C_DIS
LIN {X -0.067,Y -171.140,Z 259.378,A 0.000,B 0.000,C 90.000,E1 248.103} C_DIS
LIN {X -0.022,Y -167.444,Z 259.354,A 0.000,B 0.000,C 90.000,E1 243.768} C_DIS
LIN {X 0.061,Y -166.841,Z 259.349,A 0.000,B 0.000,C 90.000,E1 242.871} C_DIS
LIN {X -0.022,Y -162.824,Z 259.325,A 0.000,B 0.000,C 90.000,E1 238.535} C_DIS
LIN {X 0.042,Y -161.510,Z 259.315,A 0.000,B 0.000,C 90.000,E1 236.755} C_DIS
LIN {X -0.006,Y -157.508,Z 259.291,A 0.000,B 0.000,C 90.000,E1 232.351} C_DIS
LIN {X 0.028,Y -155.530,Z 259.276,A 0.000,B 0.000,C 90.000,E1 229.666} C_DIS
LIN {X 0.078,Y -151.826,Z 259.251,A 0.000,B 0.000,C 90.000,E1 225.162} C_DIS
LIN {X -0.011,Y -150.042,Z 259.236,A 0.000,B 0.000,C 90.000,E1 222.486} C_DIS
LIN {X 0.003,Y -146.857,Z 259.211,A 0.000,B 0.000,C 90.000,E1 217.935} C_DIS
LIN {X 0.021,Y -145.441,Z 259.196,A 0.000,B 0.000,C 90.000,E1 215.185} C_DIS
LIN {X 0.016,Y -142.862,Z 259.170,A 0.000,B 0.000,C 90.000,E1 210.590} C_DIS
LIN {X 0.069,Y -141.478,Z 259.149,A 0.000,B 0.000,C 90.000,E1 206.873} C_DIS
LIN {X -0.072,Y -139.381,Z 259.113,A 0.000,B 0.000,C 90.000,E1 200.429} C_DIS
LIN {X 0.049,Y -138.834,Z 259.098,A 0.000,B 0.000,C 90.000,E1 197.583} C_DIS
LIN {X -0.023,Y -138.353,Z 259.056,A 0.000,B 0.000,C 90.000,E1 190.141} C_DIS
LIN {X -0.028,Y -139.524,Z 259.004,A 0.000,B 0.000,C 90.000,E1 180.802} C_DIS
LIN {X 0.053,Y -141.193,Z 258.973,A 0.000,B 0.000,C 90.000,E1 175.184} C_DIS
LIN {X 0.024,Y -142.570,Z 258.958,A 0.000,B 0.000,C 90.000,E1 172.413} C_DIS
LIN {X -0.021,Y -144.858,Z 258.932,A 0.000,B 0.000,C 90.000,E1 167.813} C_DIS
LIN {X -0.066,Y -147.483,Z 258.912,A 0.000,B 0.000,C 90.000,E1 164.157} C_DIS
LIN {X -0.040,Y -150.070,Z 258.892,A 0.000,B 0.000,C 90.000,E1 160.496} C_DIS
LIN {X -0.036,Y -153.419,Z 258.871,A 0.000,B 0.000,C 90.000,E1 156.869} C_DIS
LIN {X 0.012,Y -156.839,Z 258.851,A 0.000,B 0.000,C 90.000,E1 153.256} C_DIS
LIN {X 0.084,Y -160.918,Z 258.832,A 0.000,B 0.000,C 90.000,E1 149.665} C_DIS
LIN {X 0.028,Y -163.044,Z 258.822,A 0.000,B 0.000,C 90.000,E1 147.916} C_DIS
LIN {X 0.033,Y -167.436,Z 258.802,A 0.000,B 0.000,C 90.000,E1 144.402} C_DIS
LIN {X -0.057,Y -171.274,Z 258.788,A 0.000,B 0.000,C 90.000,E1 141.823} C_DIS
LIN {X -0.018,Y -176.166,Z 258.769,A 0.000,B 0.000,C 90.000,E1 138.366} C_DIS
LIN {X -0.020,Y -180.437,Z 258.754,A 0.000,B 0.000,C 90.000,E1 135.810} C_DIS
LIN {X -0.046,Y -185.844,Z 258.736,A 0.000,B 0.000,C 90.000,E1 132.447} C_DIS
LIN {X 0.008,Y -190.465,Z 258.722,A 0.000,B 0.000,C 90.000,E1 129.930} C_DIS
LIN {X -0.087,Y -196.218,Z 258.704,A 0.000,B 0.000,C 90.000,E1 126.664} C_DIS
LIN {X -0.011,Y -201.028,Z 258.690,A 0.000,B 0.000,C 90.000,E1 124.199} C_DIS
LIN {X -0.030,Y -204.097,Z 258.680,A 0.000,B 0.000,C 90.000,E1 122.467} C_DIS
LIN {X -0.097,Y -307.293,Z 258.680,A 0.000,B 0.000,C 90.000,E1 122.467} C_DIS
LIN {X -0.054,Y -312.229,Z 258.679,A 0.000,B 0.000,C 90.000,E1 122.291} C_DIS
LIN {X -0.108,Y -314.606,Z 258.678,A 0.000,B 0.000,C 90.000,E1 122.133} C_DIS
LIN {X -0.116,Y -317.820,Z 258.677,A 0.000,B 0.000,C 90.000,E1 121.799} C_DIS
LIN {X 0.133,Y -319.813,Z 258.675,A 0.000,B 0.000,C 90.000,E1 121.465} C_DIS
LIN {X -0.057,Y -321.384,Z 258.673,A 0.000,B 0.000,C 90.000,E1 121.209} C_DIS
LIN {X 0.109,Y -323.965,Z 258.670,A 0.000,B 0.000,C 90.000,E1 120.541} C_DIS
LIN {X 0.019,Y -335.542,Z 258.654,A 0.000,B 0.000,C 90.000,E1 117.719} C_DIS
LIN {X -0.069,Y -348.577,Z 258.639,A 0.000,B 0.000,C 90.000,E1 114.951} C_DIS
LIN {X 0.030,Y -361.482,Z 258.625,A 0.000,B 0.000,C 90.000,E1 112.514} C_DIS
LIN {X 0.193,Y -375.725,Z 258.612,A 0.000,B 0.000,C 90.000,E1 110.120} C_DIS
LIN {X 0.110,Y -391.413,Z 258.599,A 0.000,B 0.000,C 90.000,E1 107.819} C_DIS
LIN {X -0.209,Y -408.662,Z 258.587,A 0.000,B 0.000,C 90.000,E1 105.607} C_DIS
LIN {X 0.185,Y -427.601,Z 258.574,A 0.000,B 0.000,C 90.000,E1 103.355} C_DIS
LIN {X 0.077,Y -447.713,Z 258.563,A 0.000,B 0.000,C 90.000,E1 101.299} C_DIS
LIN {X -0.190,Y -468.380,Z 258.552,A 0.000,B 0.000,C 90.000,E1 99.434} C_DIS
LIN {X -0.022,Y -492.191,Z 258.541,A 0.000,B 0.000,C 90.000,E1 97.466} C_DIS
LIN {X -0.070,Y -502.905,Z 258.537,A 0.000,B 0.000,C 90.000,E1 96.663} C_DIS
LIN {X 0.251,Y -505.001,Z 258.536,A 0.000,B 0.000,C 90.000,E1 96.429} C_DIS
LIN {X 0.211,Y -506.866,Z 258.535,A 0.000,B 0.000,C 90.000,E1 96.201} C_DIS
LIN {X 0.226,Y -508.283,Z 258.533,A 0.000,B 0.000,C 90.000,E1 95.967} C_DIS
LIN {X -0.002,Y -510.163,Z 258.531,A 0.000,B 0.000,C 90.000,E1 95.511} C_DIS
LIN {X -0.173,Y -510.898,Z 258.528,A 0.000,B 0.000,C 90.000,E1 95.049} C_DIS
LIN {X 0.174,Y -510.619,Z 258.525,A 0.000,B 0.000,C 90.000,E1 94.531} C_DIS
LIN {X -0.023,Y -509.281,Z 258.523,A 0.000,B 0.000,C 90.000,E1 94.073} C_DIS
LIN {X -0.086,Y -508.143,Z 258.521,A 0.000,B 0.000,C 90.000,E1 93.841} C_DIS
LIN {X -0.183,Y -506.613,Z 258.520,A 0.000,B 0.000,C 90.000,E1 93.612} C_DIS
LIN {X 0.031,Y -500.993,Z 258.516,A 0.000,B 0.000,C 90.000,E1 92.865} C_DIS
LIN {X 0.048,Y -492.755,Z 258.511,A 0.000,B 0.000,C 90.000,E1 91.892} C_DIS
LIN {X 0.002,Y -477.591,Z 258.501,A 0.000,B 0.000,C 90.000,E1 90.172} C_DIS
LIN {X 0.115,Y -463.198,Z 258.491,A 0.000,B 0.000,C 90.000,E1 88.396} C_DIS
LIN {X 0.189,Y -448.425,Z 258.480,A 0.000,B 0.000,C 90.000,E1 86.331} C_DIS
LIN {X 0.195,Y -428.295,Z 258.462,A 0.000,B 0.000,C 90.000,E1 83.166} C_DIS
LIN {X 0.184,Y -414.590,Z 258.449,A 0.000,B 0.000,C 90.000,E1 80.735} C_DIS
LIN {X -0.135,Y -403.280,Z 258.436,A 0.000,B 0.000,C 90.000,E1 78.578} C_DIS
LIN {X -0.088,Y -390.469,Z 258.422,A 0.000,B 0.000,C 90.000,E1 76.047} C_DIS
LIN {X 0.061,Y -379.403,Z 258.410,A 0.000,B 0.000,C 90.000,E1 73.740} C_DIS
LIN {X 0.139,Y -368.264,Z 258.397,A 0.000,B 0.000,C 90.000,E1 71.402} C_DIS
LIN {X -0.157,Y -357.344,Z 258.384,A 0.000,B 0.000,C 90.000,E1 69.082} C_DIS
LIN {X -0.042,Y -343.165,Z 258.365,A 0.000,B 0.000,C 90.000,E1 65.741} C_DIS
LIN {X -0.117,Y -331.222,Z 258.348,A 0.000,B 0.000,C 90.000,E1 62.666} C_DIS
LIN {X 0.039,Y -320.037,Z 258.331,A 0.000,B 0.000,C 90.000,E1 59.488} C_DIS
LIN {X 0.092,Y -311.279,Z 258.316,A 0.000,B 0.000,C 90.000,E1 56.914} C_DIS
LIN {X -0.144,Y -300.765,Z 258.298,A 0.000,B 0.000,C 90.000,E1 53.703} C_DIS
LIN {X 0.093,Y -292.436,Z 258.283,A 0.000,B 0.000,C 90.000,E1 51.009} C_DIS
LIN {X 0.075,Y -284.150,Z 258.269,A 0.000,B 0.000,C 90.000,E1 48.324} C_DIS
LIN {X 0.002,Y -274.156,Z 258.250,A 0.000,B 0.000,C 90.000,E1 44.919} C_DIS
LIN {X 0.068,Y -266.551,Z 258.234,A 0.000,B 0.000,C 90.000,E1 42.123} C_DIS
LIN {X -0.027,Y -259.021,Z 258.218,A 0.000,B 0.000,C 90.000,E1 39.322} C_DIS
LIN {X -0.024,Y -251.309,Z 258.203,A 0.000,B 0.000,C 90.000,E1 36.457} C_DIS
LIN {X -0.147,Y -243.613,Z 258.186,A 0.000,B 0.000,C 90.000,E1 33.579} C_DIS
LIN {X 0.005,Y -236.137,Z 258.170,A 0.000,B 0.000,C 90.000,E1 30.590} C_DIS
LIN {X 0.017,Y -229.155,Z 258.153,A 0.000,B 0.000,C 90.000,E1 27.590} C_DIS
LIN {X -0.050,Y -222.890,Z 258.136,A 0.000,B 0.000,C 90.000,E1 24.567} C_DIS
LIN {X 0.059,Y -216.093,Z 258.115,A 0.000,B 0.000,C 90.000,E1 20.684} C_DIS
LIN {X -0.027,Y -211.295,Z 258.098,A 0.000,B 0.000,C 90.000,E1 17.583} C_DIS
LIN {X -0.071,Y -206.272,Z 258.076,A 0.000,B 0.000,C 90.000,E1 13.647} C_DIS
LIN {X 0.086,Y -202.140,Z 258.054,A 0.000,B 0.000,C 90.000,E1 9.613} C_DIS
LIN {X -0.055,Y -198.619,Z 258.027,A 0.000,B 0.000,C 90.000,E1 4.821} C_DIS
LIN {X -0.077,Y -196.002,Z 257.993,A 0.000,B 0.000,C 90.000,E1 358.740} C_DIS
LIN {X 0.104,Y -197.457,Z 257.925,A 0.000,B 0.000,C 90.000,E1 346.464} C_DIS
LIN {X -0.028,Y -200.507,Z 257.898,A 0.000,B 0.000,C 90.000,E1 341.638} C_DIS
LIN {X -0.040,Y -204.262,Z 257.876,A 0.000,B 0.000,C 90.000,E1 337.614} C_DIS
LIN {X -0.106,Y -209.178,Z 257.853,A 0.000,B 0.000,C 90.000,E1 333.640} C_DIS
LIN {X -0.006,Y -215.288,Z 257.831,A 0.000,B 0.000,C 90.000,E1 329.665} C_DIS
LIN {X -0.020,Y -221.002,Z 257.814,A 0.000,B 0.000,C 90.000,E1 326.548} C_DIS
LIN {X -0.005,Y -227.659,Z 257.797,A 0.000,B 0.000,C 90.000,E1 323.463} C_DIS
LIN {X -0.057,Y -235.009,Z 257.780,A 0.000,B 0.000,C 90.000,E1 320.436} C_DIS
LIN {X -0.022,Y -244.118,Z 257.761,A 0.000,B 0.000,C 90.000,E1 317.067} C_DIS
LIN {X -0.075,Y -254.271,Z 257.743,A 0.000,B 0.000,C 90.000,E1 313.785} C_DIS
LIN {X 0.011,Y -265.502,Z 257.725,A 0.000,B 0.000,C 90.000,E1 310.539} C_DIS
LIN {X 0.114,Y -277.993,Z 257.708,A 0.000,B 0.000,C 90.000,E1 307.363} C_DIS
LIN {X 0.035,Y -288.790,Z 257.694,A 0.000,B 0.000,C 90.000,E1 304.978} C_DIS
LIN {X 0.033,Y -300.649,Z 257.681,A 0.000,B 0.000,C 90.000,E1 302.625} C_DIS
LIN {X 0.084,Y -317.565,Z 257.665,A 0.000,B 0.000,C 90.000,E1 299.667} C_DIS
LIN {X 0.113,Y -337.653,Z 257.647,A 0.000,B 0.000,C 90.000,E1 296.488} C_DIS
LIN {X 0.072,Y -350.030,Z 257.637,A 0.000,B 0.000,C 90.000,E1 294.643} C_DIS
LIN {X 0.113,Y -362.418,Z 257.627,A 0.000,B 0.000,C 90.000,E1 292.823} C_DIS
LIN {X -0.033,Y -379.211,Z 257.614,A 0.000,B 0.000,C 90.000,E1 290.482} C_DIS
LIN {X -0.031,Y -396.390,Z 257.601,A 0.000,B 0.000,C 90.000,E1 288.181} C_DIS
LIN {X -0.241,Y -407.204,Z 257.593,A 0.000,B 0.000,C 90.000,E1 286.804} C_DIS
LIN {X -0.168,Y -419.881,Z 257.584,A 0.000,B 0.000,C 90.000,E1 285.134} C_DIS
LIN {X 0.112,Y -428.126,Z 257.578,A 0.000,B 0.000,C 90.000,E1 284.008} C_DIS
LIN {X -0.107,Y -433.916,Z 257.573,A 0.000,B 0.000,C 90.000,E1 283.231} C_DIS
LIN {X 0.245,Y -441.054,Z 257.568,A 0.000,B 0.000,C 90.000,E1 282.119} C_DIS
LIN {X 0.170,Y -447.606,Z 257.562,A 0.000,B 0.000,C 90.000,E1 281.074} C_DIS
LIN {X -0.199,Y -456.862,Z 257.553,A 0.000,B 0.000,C 90.000,E1 279.557} C_DIS
LIN {X 0.196,Y -464.052,Z 257.546,A 0.000,B 0.000,C 90.000,E1 278.219} C_DIS
LIN {X 0.172,Y -470.723,Z 257.539,A 0.000,B 0.000,C 90.000,E1 276.947} C_DIS
LIN {X -0.085,Y -475.603,Z 257.533,A 0.000,B 0.000,C 90.000,E1 275.967} C_DIS
LIN {X -0.152,Y -478.829,Z 257.529,A 0.000,B 0.000,C 90.000,E1 275.220} C_DIS
LIN {X -0.005,Y -480.649,Z 257.526,A 0.000,B 0.000,C 90.000,E1 274.702} C_DIS
LIN {X 0.112,Y -482.143,Z 257.523,A 0.000,B 0.000,C 90.000,E1 274.188} C_DIS
LIN {X -0.206,Y -483.328,Z 257.521,A 0.000,B 0.000,C 90.000,E1 273.726} C_DIS
LIN {X -0.064,Y -484.155,Z 257.518,A 0.000,B 0.000,C 90.000,E1 273.212} C_DIS
LIN {X 0.112,Y -484.679,Z 257.515,A 0.000,B 0.000,C 90.000,E1 272.694} C_DIS
LIN {X -0.038,Y -485.082,Z 257.510,A 0.000,B 0.000,C 90.000,E1 271.718} C_DIS
LIN {X 0.125,Y -485.078,Z 257.507,A 0.000,B 0.000,C 90.000,E1 271.203} C_DIS
LIN {X -0.195,Y -484.895,Z 257.504,A 0.000,B 0.000,C 90.000,E1 270.745} C_DIS
LIN {X -0.029,Y -484.306,Z 257.501,A 0.000,B 0.000,C 90.000,E1 270.229} C_DIS
LIN {X 0.136,Y -483.370,Z 257.499,A 0.000,B 0.000,C 90.000,E1 269.714} C_DIS
LIN {X -0.186,Y -481.873,Z 257.496,A 0.000,B 0.000,C 90.000,E1 269.255} C_DIS
LIN {X -0.032,Y -479.754,Z 257.493,A 0.000,B 0.000,C 90.000,E1 268.740} C_DIS
LIN {X 0.111,Y -476.936,Z 257.490,A 0.000,B 0.000,C 90.000,E1 268.224} C_DIS
LIN {X -0.225,Y -473.359,Z 257.487,A 0.000,B 0.000,C 90.000,E1 267.764} C_DIS
LIN {X -0.120,Y -468.922,Z 257.485,A 0.000,B 0.000,C 90.000,E1 267.249} C_DIS
LIN {X -0.017,Y -463.581,Z 257.482,A 0.000,B 0.000,C 90.000,E1 266.731} C_DIS
LIN {X -0.089,Y -457.476,Z 257.479,A 0.000,B 0.000,C 90.000,E1 266.274} C_DIS
LIN {X 0.117,Y -454.246,Z 257.478,A 0.000,B 0.000,C 90.000,E1 266.045} C_DIS
LIN {X 0.002,Y -447.152,Z 257.476,A 0.000,B 0.000,C 90.000,E1 265.698} C_DIS
LIN {X 0.099,Y -443.032,Z 257.475,A 0.000,B 0.000,C 90.000,E1 265.527} C_DIS
LIN {X 0.068,Y -439.228,Z 257.475,A 0.000,B 0.000,C 90.000,E1 265.412} C_DIS
LIN {X 0.038,Y -434.287,Z 257.474,A 0.000,B 0.000,C 90.000,E1 265.298} C_DIS
LIN {X -0.099,Y -430.096,Z 257.473,A 0.000,B 0.000,C 90.000,E1 265.241} C_DIS
LIN {X 0.066,Y -420.810,Z 257.473,A 0.000,B 0.000,C 90.000,E1 265.122} C_DIS
LIN {X -0.014,Y -416.879,Z 257.473,A 0.000,B 0.000,C 90.000,E1 265.122} C_DIS
LIN {X -0.040,Y -180.884,Z 257.473,A 0.000,B 0.000,C 90.000,E1 265.122} C_DIS
LIN {X 0.060,Y -178.993,Z 257.444,A 0.000,B 0.000,C 90.000,E1 259.982} C_DIS
LIN {X 0.071,Y -177.983,Z 257.435,A 0.000,B 0.000,C 90.000,E1 258.285} C_DIS
LIN {X 0.041,Y -175.627,Z 257.411,A 0.000,B 0.000,C 90.000,E1 254.047} C_DIS
LIN {X 0.100,Y -172.347,Z 257.388,A 0.000,B 0.000,C 90.000,E1 249.752} C_DIS
LIN {X 0.052,Y -171.127,Z 257.378,A 0.000,B 0.000,C 90.000,E1 248.050} C_DIS
LIN {X -0.061,Y -167.435,Z 257.354,A 0.000,B 0.000,C 90.000,E1 243.768} C_DIS
LIN {X 0.022,Y -166.830,Z 257.349,A 0.000,B 0.000,C 90.000,E1 242.871} C_DIS
LIN {X -0.061,Y -162.814,Z 257.325,A 0.000,B 0.000,C 90.000,E1 238.535} C_DIS
LIN {X 0.003,Y -161.499,Z 257.315,A 0.000,B 0.000,C 90.000,E1 236.755} C_DIS
LIN {X -0.044,Y -157.497,Z 257.291,A 0.000,B 0.000,C 90.000,E1 232.351} C_DIS
LIN {X -0.009,Y -155.517,Z 257.276,A 0.000,B 0.000,C 90.000,E1 229.666} C_DIS
LIN {X 0.040,Y -151.817,Z 257.251,A 0.000,B 0.000,C 90.000,E1 225.162} C_DIS
LIN {X 0.053,Y -150.029,Z 257.236,A 0.000,B 0.000,C 90.000,E1 222.447} C_DIS
LIN {X -0.033,Y -146.849,Z 257.211,A 0.000,B 0.000,C 90.000,E1 217.935} C_DIS
LIN {X -0.014,Y -145.432,Z 257.195,A 0.000,B 0.000,C 90.000,E1 215.185} C_DIS
LIN {X -0.020,Y -142.856,Z 257.170,A 0.000,B 0.000,C 90.000,E1 210.590} C_DIS
LIN {X 0.034,Y -141.471,Z 257.149,A 0.000,B 0.000,C 90.000,E1 206.873} C_DIS
LIN {X 0.024,Y -139.379,Z 257.113,A 0.000,B 0.000,C 90.000,E1 200.375} C_DIS
LIN {X 0.015,Y -138.831,Z 257.098,A 0.000,B 0.000,C 90.000,E1 197.583} C_DIS
LIN {X -0.057,Y -138.353,Z 257.056,A 0.000,B 0.000,C 90.000,E1 190.141} C_DIS
LIN {X -0.063,Y -139.527,Z 257.004,A 0.000,B 0.000,C 90.000,E1 180.802} C_DIS
LIN {X 0.029,Y -141.199,Z 256.973,A 0.000,B 0.000,C 90.000,E1 175.179} C_DIS
LIN {X -0.011,Y -142.576,Z 256.958,A 0.000,B 0.000,C 90.000,E1 172.413} C_DIS
LIN {X -0.057,Y -144.867,Z 256.932,A 0.000,B 0.000,C 90.000,E1 167.813} C_DIS
LIN {X 0.039,Y -147.493,Z 256.912,A 0.000,B 0.000,C 90.000,E1 164.102} C_DIS
LIN {X -0.027,Y -150.082,Z 256.891,A 0.000,B 0.000,C 90.000,E1 160.477} C_DIS
LIN {X -0.013,Y -153.433,Z 256.871,A 0.000,B 0.000,C 90.000,E1 156.847} C_DIS
LIN {X -0.026,Y -156.853,Z 256.851,A 0.000,B 0.000,C 90.000,E1 153.256} C_DIS
LIN {X 0.045,Y -160.936,Z 256.832,A 0.000,B 0.000,C 90.000,E1 149.665} C_DIS
LIN {X -0.011,Y -163.059,Z 256.822,A 0.000,B 0.000,C 90.000,E1 147.916} C_DIS
LIN {X -0.006,Y -167.455,Z 256.802,A 0.000,B 0.000,C 90.000,E1 144.402} C_DIS
LIN {X 0.037,Y -171.292,Z 256.788,A 0.000,B 0.000,C 90.000,E1 141.778} C_DIS
LIN {X 0.072,Y -176.187,Z 256.769,A 0.000,B 0.000,C 90.000,E1 138.324} C_DIS
LIN {X -0.063,Y -180.462,Z 256.754,A 0.000,B 0.000,C 90.000,E1 135.810} C_DIS
LIN {X -0.088,Y -185.866,Z 256.736,A 0.000,B 0.000,C 90.000,E1 132.447} C_DIS
LIN {X -0.035,Y -190.490,Z 256.722,A 0.000,B 0.000,C 90.000,E1 129.930} C_DIS
LIN {X -0.014,Y -196.242,Z 256.703,A 0.000,B 0.000,C 90.000,E1 126.629} C_DIS
LIN {X -0.056,Y -201.048,Z 256.690,A 0.000,B 0.000,C 90.000,E1 124.199} C_DIS
LIN {X -0.032,Y -204.188,Z 256.680,A 0.000,B 0.000,C 90.000,E1 122.418} C_DIS
LIN {X -0.098,Y -307.194,Z 256.680,A 0.000,B 0.000,C 90.000,E1 122.418} C_DIS
LIN {X 0.174,Y -308.926,Z 256.680,A 0.000,B 0.000,C 90.000,E1 122.339} C_DIS
LIN {X -0.086,Y -314.696,Z 256.678,A 0.000,B 0.000,C 90.000,E1 122.084} C_DIS
LIN {X 0.085,Y -317.677,Z 256.676,A 0.000,B 0.000,C 90.000,E1 121.750} C_DIS
LIN {X 0.094,Y -319.708,Z 256.675,A 0.000,B 0.000,C 90.000,E1 121.465} C_DIS
LIN {X -0.063,Y -321.305,Z 256.673,A 0.000,B 0.000,C 90.000,E1 121.209} C_DIS
LIN {X 0.103,Y -323.948,Z 256.670,A 0.000,B 0.000,C 90.000,E1 120.541} C_DIS
LIN {X 0.012,Y -335.525,Z 256.654,A 0.000,B 0.000,C 90.000,E1 117.719} C_DIS
LIN {X -0.077,Y -348.561,Z 256.639,A 0.000,B 0.000,C 90.000,E1 114.951} C_DIS
LIN {X 0.020,Y -361.466,Z 256.625,A 0.000,B 0.000,C 90.000,E1 112.514} C_DIS
LIN {X 0.183,Y -375.711,Z 256.612,A 0.000,B 0.000,C 90.000,E1 110.120} C_DIS
LIN {X 0.100,Y -391.399,Z 256.599,A 0.000,B 0.000,C 90.000,E1 107.819} C_DIS
LIN {X -0.219,Y -408.648,Z 256.587,A 0.000,B 0.000,C 90.000,E1 105.607} C_DIS
LIN {X 0.172,Y -427.588,Z 256.574,A 0.000,B 0.000,C 90.000,E1 103.355} C_DIS
LIN {X 0.064,Y -447.700,Z 256.563,A 0.000,B 0.000,C 90.000,E1 101.299} C_DIS
LIN {X 0.259,Y -468.367,Z 256.552,A 0.000,B 0.000,C 90.000,E1 99.378} C_DIS
LIN {X -0.036,Y -492.179,Z 256.541,A 0.000,B 0.000,C 90.000,E1 97.466} C_DIS
LIN {X -0.083,Y -502.916,Z 256.537,A 0.000,B 0.000,C 90.000,E1 96.663} C_DIS
LIN {X 0.237,Y -505.069,Z 256.536,A 0.000,B 0.000,C 90.000,E1 96.429} C_DIS
LIN {X 0.230,Y -506.949,Z 256.535,A 0.000,B 0.000,C 90.000,E1 96.201} C_DIS
LIN {X 0.278,Y -508.381,Z 256.533,A 0.000,B 0.000,C 90.000,E1 95.967} C_DIS
LIN {X 0.050,Y -510.332,Z 256.531,A 0.000,B 0.000,C 90.000,E1 95.511} C_DIS
LIN {X -0.119,Y -511.132,Z 256.528,A 0.000,B 0.000,C 90.000,E1 95.049} C_DIS
LIN {X 0.228,Y -510.909,Z 256.525,A 0.000,B 0.000,C 90.000,E1 94.531} C_DIS
LIN {X 0.032,Y -509.632,Z 256.523,A 0.000,B 0.000,C 90.000,E1 94.073} C_DIS
LIN {X -0.030,Y -508.531,Z 256.521,A 0.000,B 0.000,C 90.000,E1 93.841} C_DIS
LIN {X -0.127,Y -507.044,Z 256.520,A 0.000,B 0.000,C 90.000,E1 93.612} C_DIS
LIN {X 0.090,Y -501.434,Z 256.516,A 0.000,B 0.000,C 90.000,E1 92.865} C_DIS
LIN {X 0.112,Y -493.212,Z 256.511,A 0.000,B 0.000,C 90.000,E1 91.892} C_DIS
LIN {X 0.232,Y -480.166,Z 256.502,A 0.000,B 0.000,C 90.000,E1 90.401} C_DIS
LIN {X 0.191,Y -463.580,Z 256.491,A 0.000,B 0.000,C 90.000,E1 88.396} C_DIS
LIN {X -0.176,Y -448.792,Z 256.480,A 0.000,B 0.000,C 90.000,E1 86.388} C_DIS
LIN {X 0.108,Y -430.241,Z 256.464,A 0.000,B 0.000,C 90.000,E1 83.457} C_DIS
LIN {X 0.139,Y -416.358,Z 256.450,A 0.000,B 0.000,C 90.000,E1 81.027} C_DIS
LIN {X -0.035,Y -403.557,Z 256.437,A 0.000,B 0.000,C 90.000,E1 78.578} C_DIS
LIN {X -0.076,Y -390.782,Z 256.422,A 0.000,B 0.000,C 90.000,E1 76.061} C_DIS
LIN {X 0.172,Y -379.730,Z 256.410,A 0.000,B 0.000,C 90.000,E1 73.740} C_DIS
LIN {X 0.001,Y -367.239,Z 256.395,A 0.000,B 0.000,C 90.000,E1 71.148} C_DIS
LIN {X 0.082,Y -355.064,Z 256.380,A 0.000,B 0.000,C 90.000,E1 68.465} C_DIS
LIN {X -0.059,Y -341.103,Z 256.362,A 0.000,B 0.000,C 90.000,E1 65.153} C_DIS
LIN {X 0.108,Y -329.327,Z 256.345,A 0.000,B 0.000,C 90.000,E1 62.025} C_DIS
LIN {X -0.094,Y -320.454,Z 256.331,A 0.000,B 0.000,C 90.000,E1 59.537} C_DIS
LIN {X 0.006,Y -311.705,Z 256.316,A 0.000,B 0.000,C 90.000,E1 56.962} C_DIS
LIN {X 0.039,Y -301.184,Z 256.298,A 0.000,B 0.000,C 90.000,E1 53.703} C_DIS
LIN {X -0.131,Y -292.863,Z 256.284,A 0.000,B 0.000,C 90.000,E1 51.090} C_DIS
LIN {X -0.134,Y -284.584,Z 256.269,A 0.000,B 0.000,C 90.000,E1 48.405} C_DIS
LIN {X 0.007,Y -274.571,Z 256.250,A 0.000,B 0.000,C 90.000,E1 44.960} C_DIS
LIN {X 0.092,Y -266.990,Z 256.234,A 0.000,B 0.000,C 90.000,E1 42.162} C_DIS
LIN {X -0.095,Y -261.333,Z 256.223,A 0.000,B 0.000,C 90.000,E1 40.092} C_DIS
LIN {X 0.005,Y -255.587,Z 256.211,A 0.000,B 0.000,C 90.000,E1 37.935} C_DIS
LIN {X 0.124,Y -247.900,Z 256.195,A 0.000,B 0.000,C 90.000,E1 35.025} C_DIS
LIN {X 0.003,Y -238.401,Z 256.174,A 0.000,B 0.000,C 90.000,E1 31.386} C_DIS
LIN {X -0.024,Y -231.273,Z 256.158,A 0.000,B 0.000,C 90.000,E1 28.409} C_DIS
LIN {X -0.042,Y -224.794,Z 256.141,A 0.000,B 0.000,C 90.000,E1 25.387} C_DIS
LIN {X -0.094,Y -219.115,Z 256.124,A 0.000,B 0.000,C 90.000,E1 22.333} C_DIS
LIN {X 0.026,Y -212.824,Z 256.102,A 0.000,B 0.000,C 90.000,E1 18.417} C_DIS
LIN {X 0.026,Y -207.605,Z 256.080,A 0.000,B 0.000,C 90.000,E1 14.481} C_DIS
LIN {X 0.070,Y -203.238,Z 256.058,A 0.000,B 0.000,C 90.000,E1 10.489} C_DIS
LIN {X 0.019,Y -199.415,Z 256.032,A 0.000,B 0.000,C 90.000,E1 5.682} C_DIS
LIN {X -0.035,Y -196.478,Z 255.997,A 0.000,B 0.000,C 90.000,E1 359.542} C_DIS
LIN {X -0.063,Y -197.678,Z 255.925,A 0.000,B 0.000,C 90.000,E1 346.520} C_DIS
LIN {X 0.004,Y -200.712,Z 255.898,A 0.000,B 0.000,C 90.000,E1 341.638} C_DIS
LIN {X 0.000,Y -204.459,Z 255.876,A 0.000,B 0.000,C 90.000,E1 337.614} C_DIS
LIN {X -0.059,Y -209.368,Z 255.853,A 0.000,B 0.000,C 90.000,E1 333.640} C_DIS
LIN {X 0.048,Y -215.485,Z 255.832,A 0.000,B 0.000,C 90.000,E1 329.665} C_DIS
LIN {X 0.041,Y -221.215,Z 255.814,A 0.000,B 0.000,C 90.000,E1 326.548} C_DIS
LIN {X -0.073,Y -227.881,Z 255.797,A 0.000,B 0.000,C 90.000,E1 323.497} C_DIS
LIN {X 0.019,Y -235.228,Z 255.780,A 0.000,B 0.000,C 90.000,E1 320.436} C_DIS
LIN {X 0.063,Y -244.320,Z 255.762,A 0.000,B 0.000,C 90.000,E1 317.067} C_DIS
LIN {X 0.020,Y -254.463,Z 255.743,A 0.000,B 0.000,C 90.000,E1 313.785} C_DIS
LIN {X 0.115,Y -265.662,Z 255.725,A 0.000,B 0.000,C 90.000,E1 310.539} C_DIS
LIN {X -0.162,Y -278.171,Z 255.708,A 0.000,B 0.000,C 90.000,E1 307.443} C_DIS
LIN {X -0.112,Y -290.573,Z 255.693,A 0.000,B 0.000,C 90.000,E1 304.692} C_DIS
LIN {X -0.064,Y -304.441,Z 255.678,A 0.000,B 0.000,C 90.000,E1 302.005} C_DIS
LIN {X -0.048,Y -317.731,Z 255.665,A 0.000,B 0.000,C 90.000,E1 299.716} C_DIS
LIN {X -0.031,Y -337.778,Z 255.647,A 0.000,B 0.000,C 90.000,E1 296.539} C_DIS
LIN {X -0.079,Y -350.120,Z 255.637,A 0.000,B 0.000,C 90.000,E1 294.695} C_DIS
LIN {X -0.189,Y -362.467,Z 255.627,A 0.000,B 0.000,C 90.000,E1 292.898} C_DIS
LIN {X 0.149,Y -379.192,Z 255.614,A 0.000,B 0.000,C 90.000,E1 290.482} C_DIS
LIN {X 0.159,Y -396.320,Z 255.601,A 0.000,B 0.000,C 90.000,E1 288.181} C_DIS
LIN {X 0.160,Y -409.214,Z 255.592,A 0.000,B 0.000,C 90.000,E1 286.496} C_DIS
LIN {X -0.131,Y -421.815,Z 255.583,A 0.000,B 0.000,C 90.000,E1 284.883} C_DIS
LIN {X 0.064,Y -429.970,Z 255.577,A 0.000,B 0.000,C 90.000,E1 283.772} C_DIS
LIN {X 0.045,Y -437.417,Z 255.571,A 0.000,B 0.000,C 90.000,E1 282.703} C_DIS
LIN {X -0.079,Y -444.207,Z 255.565,A 0.000,B 0.000,C 90.000,E1 281.658} C_DIS
LIN {X 0.017,Y -453.626,Z 255.556,A 0.000,B 0.000,C 90.000,E1 280.074} C_DIS
LIN {X -0.165,Y -461.026,Z 255.549,A 0.000,B 0.000,C 90.000,E1 278.803} C_DIS
LIN {X -0.230,Y -467.928,Z 255.542,A 0.000,B 0.000,C 90.000,E1 277.530} C_DIS
LIN {X -0.203,Y -474.223,Z 255.535,A 0.000,B 0.000,C 90.000,E1 276.258} C_DIS
LIN {X 0.053,Y -478.667,Z 255.529,A 0.000,B 0.000,C 90.000,E1 275.220} C_DIS
LIN {X 0.199,Y -480.511,Z 255.526,A 0.000,B 0.000,C 90.000,E1 274.702} C_DIS
LIN {X -0.165,Y -482.014,Z 255.523,A 0.000,B 0.000,C 90.000,E1 274.245} C_DIS
LIN {X -0.002,Y -483.231,Z 255.521,A 0.000,B 0.000,C 90.000,E1 273.726} C_DIS
LIN {X 0.138,Y -484.074,Z 255.518,A 0.000,B 0.000,C 90.000,E1 273.212} C_DIS
LIN {X -0.169,Y -484.641,Z 255.515,A 0.000,B 0.000,C 90.000,E1 272.751} C_DIS
LIN {X 0.164,Y -485.086,Z 255.510,A 0.000,B 0.000,C 90.000,E1 271.718} C_DIS
LIN {X 0.007,Y -484.953,Z 255.504,A 0.000,B 0.000,C 90.000,E1 270.745} C_DIS
LIN {X 0.173,Y -484.393,Z 255.501,A 0.000,B 0.000,C 90.000,E1 270.229} C_DIS
LIN {X -0.146,Y -483.497,Z 255.499,A 0.000,B 0.000,C 90.000,E1 269.771} C_DIS
LIN {X 0.016,Y -482.035,Z 255.496,A 0.000,B 0.000,C 90.000,E1 269.255} C_DIS
LIN {X 0.170,Y -479.941,Z 255.493,A 0.000,B 0.000,C 90.000,E1 268.740} C_DIS
LIN {X -0.164,Y -477.181,Z 255.490,A 0.000,B 0.000,C 90.000,E1 268.282} C_DIS
LIN {X -0.023,Y -473.656,Z 255.488,A 0.000,B 0.000,C 90.000,E1 267.764} C_DIS
LIN {X 0.081,Y -469.278,Z 255.485,A 0.000,B 0.000,C 90.000,E1 267.249} C_DIS
LIN {X 0.183,Y -464.028,Z 255.482,A 0.000,B 0.000,C 90.000,E1 266.731} C_DIS
LIN {X 0.059,Y -457.929,Z 255.479,A 0.000,B 0.000,C 90.000,E1 266.274} C_DIS
LIN {X -0.193,Y -454.803,Z 255.478,A 0.000,B 0.000,C 90.000,E1 266.102} C_DIS
LIN {X 0.041,Y -451.213,Z 255.477,A 0.000,B 0.000,C 90.000,E1 265.869} C_DIS
LIN {X 0.088,Y -447.715,Z 255.476,A 0.000,B 0.000,C 90.000,E1 265.698} C_DIS
LIN {X 0.135,Y -443.572,Z 255.475,A 0.000,B 0.000,C 90.000,E1 265.527} C_DIS
LIN {X 0.075,Y -439.737,Z 255.475,A 0.000,B 0.000,C 90.000,E1 265.412} C_DIS
LIN {X 0.015,Y -434.918,Z 255.474,A 0.000,B 0.000,C 90.000,E1 265.298} C_DIS
LIN {X -0.154,Y -430.760,Z 255.473,A 0.000,B 0.000,C 90.000,E1 265.241} C_DIS
LIN {X -0.017,Y -421.648,Z 255.473,A 0.000,B 0.000,C 90.000,E1 265.122} C_DIS
LIN {X -0.097,Y -418.980,Z 255.473,A 0.000,B 0.000,C 90.000,E1 265.122} C_DIS
LIN {X -0.076,Y -180.882,Z 255.473,A 0.000,B 0.000,C 90.000,E1 265.122} C_DIS
LIN {X 0.025,Y -178.990,Z 255.444,A 0.000,B 0.000,C 90.000,E1 259.982} C_DIS
LIN {X 0.036,Y -177.975,Z 255.435,A 0.000,B 0.000,C 90.000,E1 258.285} C_DIS
LIN {X 0.055,Y -175.619,Z 255.411,A 0.000,B 0.000,C 90.000,E1 254.031} C_DIS
LIN {X 0.066,Y -172.340,Z 255.388,A 0.000,B 0.000,C 90.000,E1 249.752} C_DIS
LIN {X 0.045,Y -171.817,Z 255.383,A 0.000,B 0.000,C 90.000,E1 248.901} C_DIS
LIN {X 0.052,Y -170.282,Z 255.373,A 0.000,B 0.000,C 90.000,E1 247.177} C_DIS
LIN {X -0.012,Y -166.822,Z 255.349,A 0.000,B 0.000,C 90.000,E1 242.871} C_DIS
LIN {X -0.094,Y -162.804,Z 255.325,A 0.000,B 0.000,C 90.000,E1 238.535} C_DIS
LIN {X -0.030,Y -161.491,Z 255.315,A 0.000,B 0.000,C 90.000,E1 236.755} C_DIS
LIN {X 0.020,Y -157.487,Z 255.291,A 0.000,B 0.000,C 90.000,E1 232.316} C_DIS
LIN {X -0.042,Y -155.505,Z 255.276,A 0.000,B 0.000,C 90.000,E1 229.666} C_DIS
LIN {X 0.009,Y -151.808,Z 255.251,A 0.000,B 0.000,C 90.000,E1 225.162} C_DIS
LIN {X 0.021,Y -150.019,Z 255.236,A 0.000,B 0.000,C 90.000,E1 222.447} C_DIS
LIN {X 0.052,Y -146.843,Z 255.211,A 0.000,B 0.000,C 90.000,E1 217.890} C_DIS
LIN {X -0.046,Y -145.425,Z 255.195,A 0.000,B 0.000,C 90.000,E1 215.185} C_DIS
LIN {X -0.050,Y -142.850,Z 255.170,A 0.000,B 0.000,C 90.000,E1 210.590} C_DIS
LIN {X 0.003,Y -141.465,Z 255.149,A 0.000,B 0.000,C 90.000,E1 206.873} C_DIS
LIN {X -0.006,Y -139.376,Z 255.113,A 0.000,B 0.000,C 90.000,E1 200.375} C_DIS
LIN {X -0.016,Y -138.827,Z 255.098,A 0.000,B 0.000,C 90.000,E1 197.583} C_DIS
LIN {X 0.048,Y -138.353,Z 255.056,A 0.000,B 0.000,C 90.000,E1 190.084} C_DIS
LIN {X 0.046,Y -139.528,Z 255.004,A 0.000,B 0.000,C 90.000,E1 180.745} C_DIS
LIN {X 0.000,Y -141.205,Z 254.973,A 0.000,B 0.000,C 90.000,E1 175.179} C_DIS
LIN {X -0.042,Y -142.580,Z 254.958,A 0.000,B 0.000,C 90.000,E1 172.413} C_DIS
LIN {X 0.054,Y -144.874,Z 254.932,A 0.000,B 0.000,C 90.000,E1 167.757} C_DIS
LIN {X 0.008,Y -147.501,Z 254.912,A 0.000,B 0.000,C 90.000,E1 164.102} C_DIS
LIN {X 0.083,Y -150.092,Z 254.891,A 0.000,B 0.000,C 90.000,E1 160.423} C_DIS
LIN {X -0.045,Y -153.446,Z 254.871,A 0.000,B 0.000,C 90.000,E1 156.847} C_DIS
LIN {X -0.051,Y -157.808,Z 254.846,A 0.000,B 0.000,C 90.000,E1 152.359} C_DIS
LIN {X -0.019,Y -162.091,Z 254.827,A 0.000,B 0.000,C 90.000,E1 148.791} C_DIS
LIN {X 0.006,Y -166.290,Z 254.807,A 0.000,B 0.000,C 90.000,E1 145.261} C_DIS
LIN {X 0.002,Y -171.308,Z 254.788,A 0.000,B 0.000,C 90.000,E1 141.778} C_DIS
LIN {X 0.037,Y -176.205,Z 254.769,A 0.000,B 0.000,C 90.000,E1 138.324} C_DIS
LIN {X -0.098,Y -180.481,Z 254.754,A 0.000,B 0.000,C 90.000,E1 135.810} C_DIS
LIN {X 0.013,Y -185.885,Z 254.736,A 0.000,B 0.000,C 90.000,E1 132.405} C_DIS
LIN {X -0.071,Y -190.511,Z 254.722,A 0.000,B 0.000,C 90.000,E1 129.930} C_DIS
LIN {X 0.107,Y -196.263,Z 254.703,A 0.000,B 0.000,C 90.000,E1 126.583} C_DIS
LIN {X -0.094,Y -201.067,Z 254.690,A 0.000,B 0.000,C 90.000,E1 124.199} C_DIS
LIN {X 0.052,Y -204.291,Z 254.680,A 0.000,B 0.000,C 90.000,E1 122.339} C_DIS
LIN {X 0.045,Y -307.415,Z 254.680,A 0.000,B 0.000,C 90.000,E1 122.339} C_DIS
LIN {X 0.037,Y -309.879,Z 254.679,A 0.000,B 0.000,C 90.000,E1 122.291} C_DIS
LIN {X 0.114,Y -314.750,Z 254.678,A 0.000,B 0.000,C 90.000,E1 122.005} C_DIS
LIN {X 0.025,Y -317.505,Z 254.676,A 0.000,B 0.000,C 90.000,E1 121.750} C_DIS
LIN {X -0.048,Y -321.196,Z 254.673,A 0.000,B 0.000,C 90.000,E1 121.209} C_DIS
LIN {X 0.029,Y -322.693,Z 254.672,A 0.000,B 0.000,C 90.000,E1 120.875} C_DIS
LIN {X 0.045,Y -334.147,Z 254.656,A 0.000,B 0.000,C 90.000,E1 118.025} C_DIS
LIN {X 0.081,Y -347.012,Z 254.640,A 0.000,B 0.000,C 90.000,E1 115.232} C_DIS
LIN {X -0.031,Y -359.756,Z 254.627,A 0.000,B 0.000,C 90.000,E1 112.823} C_DIS
LIN {X 0.085,Y -373.826,Z 254.614,A 0.000,B 0.000,C 90.000,E1 110.429} C_DIS
LIN {X -0.046,Y -389.327,Z 254.601,A 0.000,B 0.000,C 90.000,E1 108.127} C_DIS
LIN {X 0.087,Y -406.375,Z 254.588,A 0.000,B 0.000,C 90.000,E1 105.843} C_DIS
LIN {X 0.020,Y -425.095,Z 254.576,A 0.000,B 0.000,C 90.000,E1 103.647} C_DIS
LIN {X 0.173,Y -445.116,Z 254.564,A 0.000,B 0.000,C 90.000,E1 101.535} C_DIS
LIN {X 0.204,Y -465.718,Z 254.554,A 0.000,B 0.000,C 90.000,E1 99.613} C_DIS
LIN {X 0.203,Y -489.495,Z 254.543,A 0.000,B 0.000,C 90.000,E1 97.644} C_DIS
LIN {X -0.088,Y -502.908,Z 254.537,A 0.000,B 0.000,C 90.000,E1 96.663} C_DIS
LIN {X 0.232,Y -505.127,Z 254.536,A 0.000,B 0.000,C 90.000,E1 96.429} C_DIS
LIN {X -0.242,Y -507.025,Z 254.535,A 0.000,B 0.000,C 90.000,E1 96.258} C_DIS
LIN {X -0.160,Y -508.473,Z 254.533,A 0.000,B 0.000,C 90.000,E1 96.024} C_DIS
LIN {X 0.119,Y -510.492,Z 254.531,A 0.000,B 0.000,C 90.000,E1 95.511} C_DIS
LIN {X -0.050,Y -511.346,Z 254.528,A 0.000,B 0.000,C 90.000,E1 95.049} C_DIS
LIN {X -0.211,Y -511.181,Z 254.525,A 0.000,B 0.000,C 90.000,E1 94.588} C_DIS
LIN {X 0.103,Y -509.967,Z 254.523,A 0.000,B 0.000,C 90.000,E1 94.073} C_DIS
LIN {X 0.042,Y -508.905,Z 254.521,A 0.000,B 0.000,C 90.000,E1 93.841} C_DIS
LIN {X -0.055,Y -507.465,Z 254.520,A 0.000,B 0.000,C 90.000,E1 93.612} C_DIS
LIN {X 0.056,Y -499.921,Z 254.515,A 0.000,B 0.000,C 90.000,E1 92.636} C_DIS
LIN {X -0.060,Y -489.389,Z 254.508,A 0.000,B 0.000,C 90.000,E1 91.432} C_DIS
LIN {X 0.020,Y -465.959,Z 254.493,A 0.000,B 0.000,C 90.000,E1 88.682} C_DIS
LIN {X -0.085,Y -452.762,Z 254.483,A 0.000,B 0.000,C 90.000,E1 86.906} C_DIS
LIN {X 0.160,Y -435.510,Z 254.468,A 0.000,B 0.000,C 90.000,E1 84.261} C_DIS
LIN {X 0.108,Y -418.157,Z 254.452,A 0.000,B 0.000,C 90.000,E1 81.319} C_DIS
LIN {X -0.028,Y -405.283,Z 254.438,A 0.000,B 0.000,C 90.000,E1 78.870} C_DIS
LIN {X -0.087,Y -393.906,Z 254.426,A 0.000,B 0.000,C 90.000,E1 76.645} C_DIS
LIN {X -0.196,Y -381.428,Z 254.412,A 0.000,B 0.000,C 90.000,E1 74.102} C_DIS
LIN {X -0.054,Y -371.712,Z 254.400,A 0.000,B 0.000,C 90.000,E1 72.054} C_DIS
LIN {X -0.042,Y -360.806,Z 254.387,A 0.000,B 0.000,C 90.000,E1 69.699} C_DIS
LIN {X 0.183,Y -346.439,Z 254.369,A 0.000,B 0.000,C 90.000,E1 66.357} C_DIS
LIN {X 0.034,Y -333.217,Z 254.350,A 0.000,B 0.000,C 90.000,E1 62.999} C_DIS
LIN {X 0.061,Y -320.855,Z 254.331,A 0.000,B 0.000,C 90.000,E1 59.537} C_DIS
LIN {X -0.003,Y -312.116,Z 254.317,A 0.000,B 0.000,C 90.000,E1 56.993} C_DIS
LIN {X -0.036,Y -301.611,Z 254.299,A 0.000,B 0.000,C 90.000,E1 53.749} C_DIS
LIN {X 0.043,Y -293.280,Z 254.284,A 0.000,B 0.000,C 90.000,E1 51.090} C_DIS
LIN {X 0.044,Y -285.012,Z 254.269,A 0.000,B 0.000,C 90.000,E1 48.405} C_DIS
LIN {X -0.001,Y -274.989,Z 254.250,A 0.000,B 0.000,C 90.000,E1 45.000} C_DIS
LIN {X 0.087,Y -267.426,Z 254.235,A 0.000,B 0.000,C 90.000,E1 42.204} C_DIS
LIN {X 0.100,Y -261.774,Z 254.223,A 0.000,B 0.000,C 90.000,E1 40.092} C_DIS
LIN {X -0.077,Y -254.090,Z 254.207,A 0.000,B 0.000,C 90.000,E1 37.282} C_DIS
LIN {X -0.137,Y -246.415,Z 254.191,A 0.000,B 0.000,C 90.000,E1 34.405} C_DIS
LIN {X 0.113,Y -236.980,Z 254.171,A 0.000,B 0.000,C 90.000,E1 30.669} C_DIS
LIN {X -0.001,Y -228.369,Z 254.150,A 0.000,B 0.000,C 90.000,E1 26.950} C_DIS
LIN {X 0.023,Y -222.270,Z 254.133,A 0.000,B 0.000,C 90.000,E1 23.898} C_DIS
LIN {X -0.082,Y -215.641,Z 254.111,A 0.000,B 0.000,C 90.000,E1 20.066} C_DIS
LIN {X -0.009,Y -209.958,Z 254.090,A 0.000,B 0.000,C 90.000,E1 16.134} C_DIS
LIN {X -0.008,Y -205.206,Z 254.068,A 0.000,B 0.000,C 90.000,E1 12.175} C_DIS
LIN {X 0.062,Y -200.843,Z 254.041,A 0.000,B 0.000,C 90.000,E1 7.352} C_DIS
LIN {X -0.011,Y -197.532,Z 254.010,A 0.000,B 0.000,C 90.000,E1 1.718} C_DIS
LIN {X -0.011,Y -198.295,Z 253.921,A 0.000,B 0.000,C 90.000,E1 345.700} C_DIS
LIN {X -0.062,Y -201.563,Z 253.894,A 0.000,B 0.000,C 90.000,E1 340.859} C_DIS
LIN {X 0.108,Y -205.559,Z 253.871,A 0.000,B 0.000,C 90.000,E1 336.794} C_DIS
LIN {X -0.101,Y -210.698,Z 253.849,A 0.000,B 0.000,C 90.000,E1 332.871} C_DIS
LIN {X -0.032,Y -217.036,Z 253.827,A 0.000,B 0.000,C 90.000,E1 328.918} C_DIS
LIN {X 0.000,Y -223.027,Z 253.810,A 0.000,B 0.000,C 90.000,E1 325.801} C_DIS
LIN {X 0.061,Y -229.871,Z 253.793,A 0.000,B 0.000,C 90.000,E1 322.718} C_DIS
LIN {X 0.020,Y -237.388,Z 253.776,A 0.000,B 0.000,C 90.000,E1 319.703} C_DIS
LIN {X -0.053,Y -246.661,Z 253.758,A 0.000,B 0.000,C 90.000,E1 316.377} C_DIS
LIN {X -0.030,Y -256.992,Z 253.739,A 0.000,B 0.000,C 90.000,E1 313.095} C_DIS
LIN {X -0.031,Y -268.499,Z 253.722,A 0.000,B 0.000,C 90.000,E1 309.886} C_DIS
LIN {X -0.006,Y -281.332,Z 253.704,A 0.000,B 0.000,C 90.000,E1 306.744} C_DIS
LIN {X 0.158,Y -292.376,Z 253.691,A 0.000,B 0.000,C 90.000,E1 304.326} C_DIS
LIN {X 0.097,Y -306.448,Z 253.676,A 0.000,B 0.000,C 90.000,E1 301.671} C_DIS
LIN {X 0.077,Y -321.772,Z 253.662,A 0.000,B 0.000,C 90.000,E1 299.077} C_DIS
LIN {X 0.103,Y -339.957,Z 253.646,A 0.000,B 0.000,C 90.000,E1 296.232} C_DIS
LIN {X 0.103,Y -352.236,Z 253.636,A 0.000,B 0.000,C 90.000,E1 294.387} C_DIS
LIN {X 0.044,Y -364.564,Z 253.626,A 0.000,B 0.000,C 90.000,E1 292.589} C_DIS
LIN {X 0.082,Y -383.422,Z 253.611,A 0.000,B 0.000,C 90.000,E1 289.939} C_DIS
LIN {X 0.197,Y -400.558,Z 253.598,A 0.000,B 0.000,C 90.000,E1 287.638} C_DIS
LIN {X 0.053,Y -411.223,Z 253.590,A 0.000,B 0.000,C 90.000,E1 286.260} C_DIS
LIN {X 0.204,Y -423.785,Z 253.581,A 0.000,B 0.000,C 90.000,E1 284.592} C_DIS
LIN {X 0.013,Y -431.721,Z 253.575,A 0.000,B 0.000,C 90.000,E1 283.536} C_DIS
LIN {X 0.150,Y -437.244,Z 253.571,A 0.000,B 0.000,C 90.000,E1 282.715} C_DIS
LIN {X 0.123,Y -444.042,Z 253.565,A 0.000,B 0.000,C 90.000,E1 281.658} C_DIS
LIN {X 0.141,Y -453.437,Z 253.556,A 0.000,B 0.000,C 90.000,E1 280.084} C_DIS
LIN {X 0.040,Y -460.802,Z 253.549,A 0.000,B 0.000,C 90.000,E1 278.803} C_DIS
LIN {X 0.201,Y -466.384,Z 253.543,A 0.000,B 0.000,C 90.000,E1 277.757} C_DIS
LIN {X 0.211,Y -472.796,Z 253.536,A 0.000,B 0.000,C 90.000,E1 276.486} C_DIS
LIN {X -0.072,Y -477.429,Z 253.531,A 0.000,B 0.000,C 90.000,E1 275.511} C_DIS
LIN {X -0.076,Y -480.371,Z 253.526,A 0.000,B 0.000,C 90.000,E1 274.759} C_DIS
LIN {X 0.038,Y -481.910,Z 253.524,A 0.000,B 0.000,C 90.000,E1 274.245} C_DIS
LIN {X 0.200,Y -483.129,Z 253.521,A 0.000,B 0.000,C 90.000,E1 273.726} C_DIS
LIN {X -0.143,Y -484.023,Z 253.518,A 0.000,B 0.000,C 90.000,E1 273.269} C_DIS
LIN {X 0.032,Y -484.599,Z 253.515,A 0.000,B 0.000,C 90.000,E1 272.751} C_DIS
LIN {X -0.119,Y -485.120,Z 253.510,A 0.000,B 0.000,C 90.000,E1 271.776} C_DIS
LIN {X 0.043,Y -485.149,Z 253.507,A 0.000,B 0.000,C 90.000,E1 271.260} C_DIS
LIN {X 0.209,Y -485.002,Z 253.504,A 0.000,B 0.000,C 90.000,E1 270.745} C_DIS
LIN {X -0.109,Y -484.462,Z 253.502,A 0.000,B 0.000,C 90.000,E1 270.286} C_DIS
LIN {X 0.056,Y -483.586,Z 253.499,A 0.000,B 0.000,C 90.000,E1 269.771} C_DIS
LIN {X 0.218,Y -482.170,Z 253.496,A 0.000,B 0.000,C 90.000,E1 269.255} C_DIS
LIN {X -0.109,Y -480.106,Z 253.493,A 0.000,B 0.000,C 90.000,E1 268.797} C_DIS
LIN {X 0.037,Y -477.407,Z 253.490,A 0.000,B 0.000,C 90.000,E1 268.282} C_DIS
LIN {X 0.177,Y -473.946,Z 253.488,A 0.000,B 0.000,C 90.000,E1 267.764} C_DIS
LIN {X -0.188,Y -469.624,Z 253.485,A 0.000,B 0.000,C 90.000,E1 267.306} C_DIS
LIN {X 0.086,Y -467.189,Z 253.484,A 0.000,B 0.000,C 90.000,E1 267.020} C_DIS
LIN {X -0.132,Y -461.653,Z 253.481,A 0.000,B 0.000,C 90.000,E1 266.560} C_DIS
LIN {X -0.182,Y -458.547,Z 253.479,A 0.000,B 0.000,C 90.000,E1 266.331} C_DIS
LIN {X 0.195,Y -451.852,Z 253.477,A 0.000,B 0.000,C 90.000,E1 265.869} C_DIS
LIN {X 0.204,Y -448.377,Z 253.476,A 0.000,B 0.000,C 90.000,E1 265.698} C_DIS
LIN {X 0.212,Y -444.236,Z 253.475,A 0.000,B 0.000,C 90.000,E1 265.527} C_DIS
LIN {X 0.126,Y -440.435,Z 253.475,A 0.000,B 0.000,C 90.000,E1 265.412} C_DIS
LIN {X -0.156,Y -431.725,Z 253.473,A 0.000,B 0.000,C 90.000,E1 265.241} C_DIS
LIN {X -0.145,Y -421.257,Z 253.473,A 0.000,B 0.000,C 90.000,E1 265.122} C_DIS
LIN {X 0.187,Y -416.128,Z 253.473,A 0.000,B 0.000,C 90.000,E1 265.065} C_DIS
LIN {X 0.063,Y -180.879,Z 253.473,A 0.000,B 0.000,C 90.000,E1 265.065} C_DIS
LIN {X -0.008,Y -178.987,Z 253.444,A 0.000,B 0.000,C 90.000,E1 259.982} C_DIS
LIN {X 0.003,Y -177.968,Z 253.435,A 0.000,B 0.000,C 90.000,E1 258.285} C_DIS
LIN {X 0.022,Y -175.611,Z 253.411,A 0.000,B 0.000,C 90.000,E1 254.031} C_DIS
LIN {X 0.035,Y -172.333,Z 253.388,A 0.000,B 0.000,C 90.000,E1 249.752} C_DIS
LIN {X 0.013,Y -171.810,Z 253.383,A 0.000,B 0.000,C 90.000,E1 248.901} C_DIS
LIN {X 0.021,Y -170.273,Z 253.373,A 0.000,B 0.000,C 90.000,E1 247.177} C_DIS
LIN {X -0.043,Y -166.814,Z 253.349,A 0.000,B 0.000,C 90.000,E1 242.871} C_DIS
LIN {X 0.014,Y -162.796,Z 253.325,A 0.000,B 0.000,C 90.000,E1 238.486} C_DIS
LIN {X 0.074,Y -161.483,Z 253.315,A 0.000,B 0.000,C 90.000,E1 236.707} C_DIS
LIN {X -0.010,Y -157.479,Z 253.291,A 0.000,B 0.000,C 90.000,E1 232.316} C_DIS
LIN {X 0.046,Y -155.495,Z 253.276,A 0.000,B 0.000,C 90.000,E1 229.622} C_DIS
LIN {X -0.021,Y -151.801,Z 253.251,A 0.000,B 0.000,C 90.000,E1 225.162} C_DIS
LIN {X -0.008,Y -150.011,Z 253.236,A 0.000,B 0.000,C 90.000,E1 222.447} C_DIS
LIN {X 0.022,Y -146.836,Z 253.211,A 0.000,B 0.000,C 90.000,E1 217.890} C_DIS
LIN {X 0.009,Y -145.417,Z 253.195,A 0.000,B 0.000,C 90.000,E1 215.152} C_DIS
LIN {X 0.044,Y -142.845,Z 253.170,A 0.000,B 0.000,C 90.000,E1 210.541} C_DIS
LIN {X -0.025,Y -141.459,Z 253.149,A 0.000,B 0.000,C 90.000,E1 206.873} C_DIS
LIN {X 0.015,Y -139.374,Z 253.113,A 0.000,B 0.000,C 90.000,E1 200.355} C_DIS
LIN {X -0.043,Y -138.825,Z 253.098,A 0.000,B 0.000,C 90.000,E1 197.583} C_DIS
LIN {X 0.045,Y -138.353,Z 253.056,A 0.000,B 0.000,C 90.000,E1 190.074} C_DIS
LIN {X 0.018,Y -139.531,Z 253.004,A 0.000,B 0.000,C 90.000,E1 180.745} C_DIS
LIN {X -0.029,Y -141.210,Z 252.973,A 0.000,B 0.000,C 90.000,E1 175.179} C_DIS
LIN {X 0.071,Y -142.585,Z 252.958,A 0.000,B 0.000,C 90.000,E1 172.356} C_DIS
LIN {X 0.025,Y -144.881,Z 252.932,A 0.000,B 0.000,C 90.000,E1 167.757} C_DIS
LIN {X -0.021,Y -147.508,Z 252.912,A 0.000,B 0.000,C 90.000,E1 164.102} C_DIS
LIN {X 0.053,Y -150.101,Z 252.891,A 0.000,B 0.000,C 90.000,E1 160.423} C_DIS
LIN {X 0.066,Y -153.458,Z 252.871,A 0.000,B 0.000,C 90.000,E1 156.794} C_DIS
LIN {X -0.082,Y -157.821,Z 252.846,A 0.000,B 0.000,C 90.000,E1 152.359} C_DIS
LIN {X -0.050,Y -162.104,Z 252.827,A 0.000,B 0.000,C 90.000,E1 148.791} C_DIS
LIN {X -0.026,Y -166.304,Z 252.807,A 0.000,B 0.000,C 90.000,E1 145.261} C_DIS
LIN {X -0.030,Y -171.322,Z 252.788,A 0.000,B 0.000,C 90.000,E1 141.778} C_DIS
LIN {X 0.005,Y -176.221,Z 252.768,A 0.000,B 0.000,C 90.000,E1 138.324} C_DIS
LIN {X -0.002,Y -180.500,Z 252.754,A 0.000,B 0.000,C 90.000,E1 135.769} C_DIS
LIN {X -0.020,Y -185.903,Z 252.736,A 0.000,B 0.000,C 90.000,E1 132.405} C_DIS
LIN {X 0.040,Y -190.531,Z 252.722,A 0.000,B 0.000,C 90.000,E1 129.886} C_DIS
LIN {X 0.072,Y -196.281,Z 252.703,A 0.000,B 0.000,C 90.000,E1 126.583} C_DIS
LIN {X -0.128,Y -201.084,Z 252.690,A 0.000,B 0.000,C 90.000,E1 124.199} C_DIS
LIN {X 0.053,Y -204.381,Z 252.679,A 0.000,B 0.000,C 90.000,E1 122.291} C_DIS
LIN {X 0.031,Y -307.413,Z 252.679,A 0.000,B 0.000,C 90.000,E1 122.291} C_DIS
LIN {X -0.019,Y -308.235,Z 252.679,A 0.000,B 0.000,C 90.000,E1 122.291} C_DIS
LIN {X 0.059,Y -314.372,Z 252.678,A 0.000,B 0.000,C 90.000,E1 122.005} C_DIS
LIN {X -0.029,Y -317.297,Z 252.676,A 0.000,B 0.000,C 90.000,E1 121.750} C_DIS
LIN {X 0.040,Y -321.000,Z 252.673,A 0.000,B 0.000,C 90.000,E1 121.209} C_DIS
LIN {X 0.115,Y -322.579,Z 252.672,A 0.000,B 0.000,C 90.000,E1 120.875} C_DIS
LIN {X 0.100,Y -335.414,Z 252.654,A 0.000,B 0.000,C 90.000,E1 117.719} C_DIS
LIN {X 0.011,Y -348.443,Z 252.639,A 0.000,B 0.000,C 90.000,E1 114.951} C_DIS
LIN {X 0.110,Y -361.338,Z 252.625,A 0.000,B 0.000,C 90.000,E1 112.514} C_DIS
LIN {X -0.080,Y -375.574,Z 252.612,A 0.000,B 0.000,C 90.000,E1 110.174} C_DIS
LIN {X 0.189,Y -391.253,Z 252.599,A 0.000,B 0.000,C 90.000,E1 107.819} C_DIS
LIN {X -0.130,Y -408.493,Z 252.587,A 0.000,B 0.000,C 90.000,E1 105.607} C_DIS
LIN {X -0.154,Y -427.422,Z 252.574,A 0.000,B 0.000,C 90.000,E1 103.411} C_DIS
LIN {X 0.148,Y -447.532,Z 252.563,A 0.000,B 0.000,C 90.000,E1 101.299} C_DIS
LIN {X -0.125,Y -468.196,Z 252.552,A 0.000,B 0.000,C 90.000,E1 99.434} C_DIS
LIN {X 0.037,Y -492.005,Z 252.542,A 0.000,B 0.000,C 90.000,E1 97.466} C_DIS
LIN {X -0.012,Y -502.766,Z 252.537,A 0.000,B 0.000,C 90.000,E1 96.663} C_DIS
LIN {X -0.195,Y -505.082,Z 252.536,A 0.000,B 0.000,C 90.000,E1 96.486} C_DIS
LIN {X -0.031,Y -508.477,Z 252.533,A 0.000,B 0.000,C 90.000,E1 96.030} C_DIS
LIN {X -0.098,Y -509.711,Z 252.532,A 0.000,B 0.000,C 90.000,E1 95.796} C_DIS
LIN {X -0.219,Y -510.606,Z 252.531,A 0.000,B 0.000,C 90.000,E1 95.568} C_DIS
LIN {X 0.127,Y -511.541,Z 252.528,A 0.000,B 0.000,C 90.000,E1 95.049} C_DIS
LIN {X -0.032,Y -511.457,Z 252.525,A 0.000,B 0.000,C 90.000,E1 94.588} C_DIS
LIN {X -0.226,Y -510.332,Z 252.523,A 0.000,B 0.000,C 90.000,E1 94.131} C_DIS
LIN {X 0.222,Y -509.323,Z 252.521,A 0.000,B 0.000,C 90.000,E1 93.841} C_DIS
LIN {X 0.125,Y -507.949,Z 252.520,A 0.000,B 0.000,C 90.000,E1 93.612} C_DIS
LIN {X -0.154,Y -502.422,Z 252.516,A 0.000,B 0.000,C 90.000,E1 92.922} C_DIS
LIN {X -0.118,Y -494.243,Z 252.511,A 0.000,B 0.000,C 90.000,E1 91.949} C_DIS
LIN {X 0.183,Y -483.376,Z 252.504,A 0.000,B 0.000,C 90.000,E1 90.688} C_DIS
LIN {X 0.215,Y -466.471,Z 252.493,A 0.000,B 0.000,C 90.000,E1 88.682} C_DIS
LIN {X -0.110,Y -455.043,Z 252.484,A 0.000,B 0.000,C 90.000,E1 87.192} C_DIS
LIN {X 0.167,Y -437.604,Z 252.470,A 0.000,B 0.000,C 90.000,E1 84.552} C_DIS
LIN {X 0.226,Y -420.052,Z 252.454,A 0.000,B 0.000,C 90.000,E1 81.602} C_DIS
LIN {X -0.102,Y -404.237,Z 252.437,A 0.000,B 0.000,C 90.000,E1 78.634} C_DIS
LIN {X -0.119,Y -391.491,Z 252.423,A 0.000,B 0.000,C 90.000,E1 76.117} C_DIS
LIN {X 0.152,Y -380.444,Z 252.410,A 0.000,B 0.000,C 90.000,E1 73.795} C_DIS
LIN {X -0.112,Y -368.025,Z 252.396,A 0.000,B 0.000,C 90.000,E1 71.221} C_DIS
LIN {X -0.016,Y -355.912,Z 252.381,A 0.000,B 0.000,C 90.000,E1 68.539} C_DIS
LIN {X -0.129,Y -340.762,Z 252.361,A 0.000,B 0.000,C 90.000,E1 64.921} C_DIS
END
